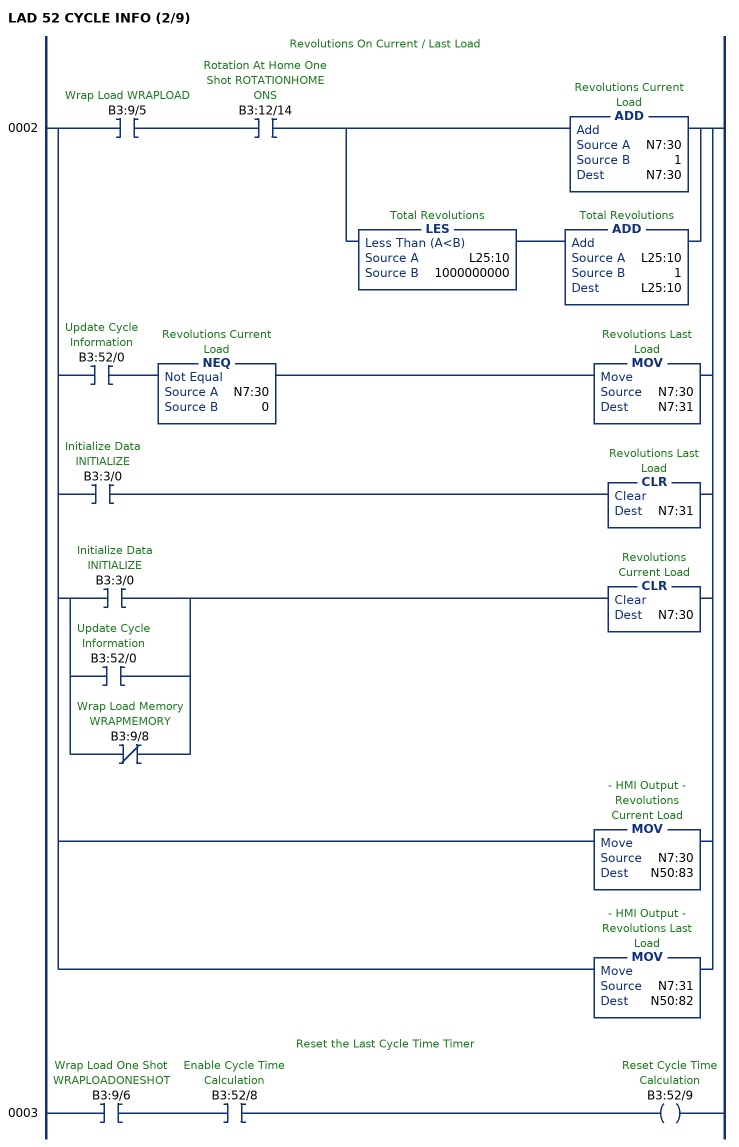
% Rung: 2 %
% Revolutions On Current / Last Load %
SOR BST XIC B3:9/5 XIC B3:12/14 BST ADD N7:30 1 N7:30 NXB LES L25:10 1000000000 ADD L25:10 1 L25:10 BND NXB XIC B3:52/0 NEQ N7:30 0 MOV N7:30 N7:31 NXB XIC B3:3/0 CLR N7:31 NXB BST XIC B3:3/0 NXB XIC B3:52/0 NXB XIO B3:9/8 BND CLR N7:30 NXB MOV N7:30 N50:83 NXB MOV N7:31 N50:82 BND EOR
%   B3:9/5  WRAPLOAD  "Wrap Load" %
%   B3:12/14  ROTATIONHOMEONS  "Rotation At Home One Shot" %
%   N7:30  "Revolutions Current Load" %
%   L25:10  "Total Revolutions" %
%   B3:52/0  "Update Cycle Information" %
%   N7:31  "Revolutions Last Load" %
%   B3:3/0  INITIALIZE  "Initialize Data" %
%   B3:9/8  WRAPMEMORY  "Wrap Load Memory" %
%   N50:83  "- HMI Output - Revolutions Current Load" %
%   N50:82  "- HMI Output - Revolutions Last Load" %
% Rung: 3 %
% Reset the Last Cycle Time Timer %
SOR XIC B3:9/6 XIC B3:52/8 OTE B3:52/9 EOR
%   B3:9/6  WRAPLOADONESHOT  "Wrap Load One Shot" %
%   B3:52/8  "Enable Cycle Time Calculation" %
%   B3:52/9  "Reset Cycle Time Calculation" %

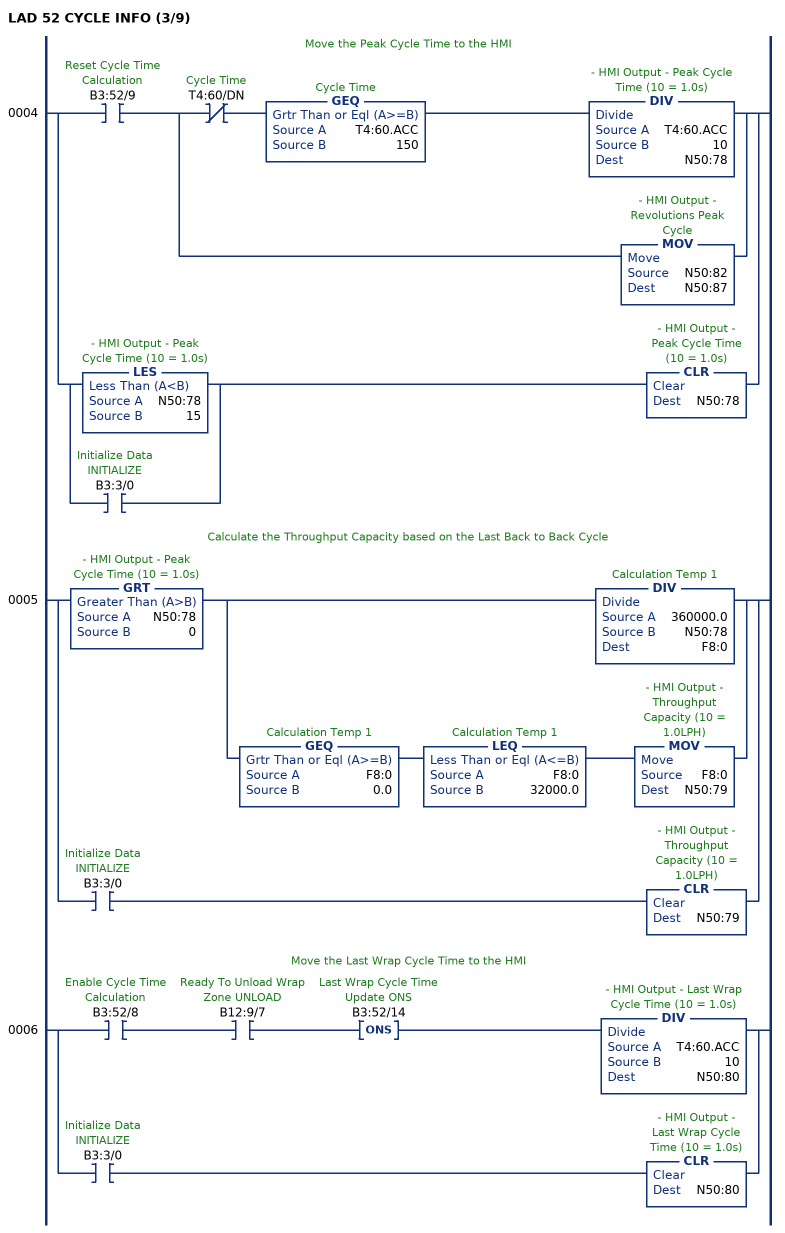
% Rung: 4 %
% Move the Peak Cycle Time to the HMI %
SOR BST XIC B3:52/9 BST XIO T4:60/DN GEQ T4:60.ACC 150 DIV T4:60.ACC 10 N50:78 NXB MOV N50:82 N50:87 BND NXB BST LES N50:78 15 NXB XIC B3:3/0 BND CLR N50:78 BND EOR
%   B3:52/9  "Reset Cycle Time Calculation" %
%   T4:60  "Cycle Time" %
%   N50:78  "- HMI Output - Peak Cycle Time (10 = 1.0s)" %
%   N50:82  "- HMI Output - Revolutions Last Load" %
%   N50:87  "- HMI Output - Revolutions Peak Cycle" %
%   B3:3/0  INITIALIZE  "Initialize Data" %
% Rung: 5 %
% Calculate the Throughput Capacity based on the Last Back to Back Cycle %
SOR BST GRT N50:78 0 BST DIV 360000.0 N50:78 F8:0 NXB GEQ F8:0 0.0 LEQ F8:0 32000.0 MOV F8:0 N50:79 BND NXB XIC B3:3/0 CLR N50:79 BND EOR
%   N50:78  "- HMI Output - Peak Cycle Time (10 = 1.0s)" %
%   F8:0  "Calculation Temp 1" %
%   N50:79  "- HMI Output - Throughput Capacity (10 = 1.0LPH)" %
%   B3:3/0  INITIALIZE  "Initialize Data" %
% Rung: 6 %
% Move the Last Wrap Cycle Time to the HMI %
SOR BST XIC B3:52/8 XIC B12:9/7 ONS B3:52/14 DIV T4:60.ACC 10 N50:80 NXB XIC B3:3/0 CLR N50:80 BND EOR
%   B3:52/8  "Enable Cycle Time Calculation" %
%   B12:9/7  UNLOAD  "Ready To Unload Wrap Zone" %
%   B3:52/14  "Last Wrap Cycle Time Update ONS" %
%   T4:60  "Cycle Time" %
%   N50:80  "- HMI Output - Last Wrap Cycle Time (10 = 1.0s)" %
%   B3:3/0  INITIALIZE  "Initialize Data" %

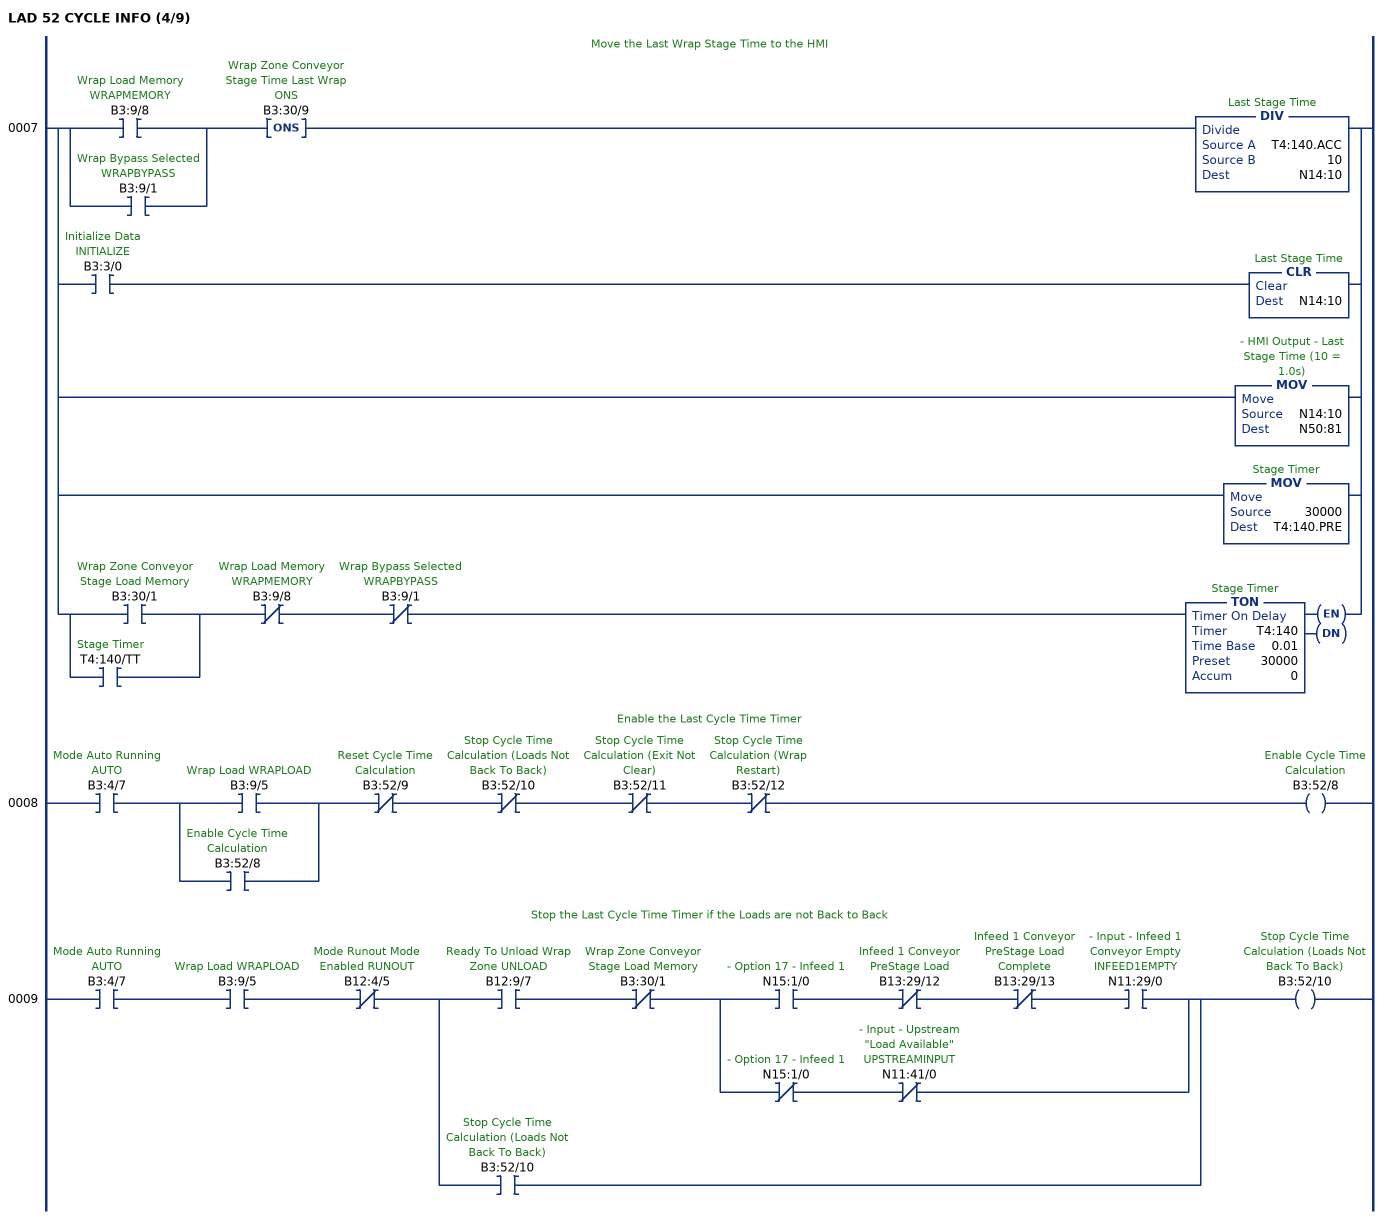
% Rung: 7 %
% Move the Last Wrap Stage Time to the HMI %
SOR BST BST XIC B3:9/8 NXB XIC B3:9/1 BND ONS B3:30/9 DIV T4:140.ACC 10 N14:10 NXB XIC B3:3/0 CLR N14:10 NXB MOV N14:10 N50:81 NXB MOV 30000 T4:140.PRE NXB BST XIC B3:30/1 NXB XIC T4:140/TT BND XIO B3:9/8 XIO B3:9/1 TON T4:140 0.01 30000 0 BND EOR
%   B3:9/8  WRAPMEMORY  "Wrap Load Memory" %
%   B3:9/1  WRAPBYPASS  "Wrap Bypass Selected" %
%   B3:30/9  "Wrap Zone Conveyor Stage Time Last Wrap ONS" %
%   T4:140  "Stage Timer" %
%   N14:10  "Last Stage Time" %
%   B3:3/0  INITIALIZE  "Initialize Data" %
%   N50:81  "- HMI Output - Last Stage Time (10 = 1.0s)" %
%   B3:30/1  "Wrap Zone Conveyor Stage Load Memory" %
% Rung: 8 %
% Enable the Last Cycle Time Timer %
SOR XIC B3:4/7 BST XIC B3:9/5 NXB XIC B3:52/8 BND XIO B3:52/9 XIO B3:52/10 XIO B3:52/11 XIO B3:52/12 OTE B3:52/8 EOR
%   B3:4/7  AUTO  "Mode Auto Running" %
%   B3:9/5  WRAPLOAD  "Wrap Load" %
%   B3:52/8  "Enable Cycle Time Calculation" %
%   B3:52/9  "Reset Cycle Time Calculation" %
%   B3:52/10  "Stop Cycle Time Calculation (Loads Not Back To Back)" %
%   B3:52/11  "Stop Cycle Time Calculation (Exit Not Clear)" %
%   B3:52/12  "Stop Cycle Time Calculation (Wrap Restart)" %
% Rung: 9 %
% Stop the Last Cycle Time Timer if the Loads are not Back to Back %
SOR XIC B3:4/7 XIC B3:9/5 XIO B12:4/5 BST XIC B12:9/7 XIO B3:30/1 BST XIC N15:1/0 XIO B13:29/12 XIO B13:29/13 XIC N11:29/0 NXB XIO N15:1/0 XIO N11:41/0 BND NXB XIC B3:52/10 BND OTE B3:52/10 EOR
%   B3:4/7  AUTO  "Mode Auto Running" %
%   B3:9/5  WRAPLOAD  "Wrap Load" %
%   B12:4/5  RUNOUT  "Mode Runout Mode Enabled" %
%   B12:9/7  UNLOAD  "Ready To Unload Wrap Zone" %
%   B3:30/1  "Wrap Zone Conveyor Stage Load Memory" %
%   N15:1/0  "- Option 17 - Infeed 1" %
%   B13:29/12  "Infeed 1 Conveyor PreStage Load" %
%   B13:29/13  "Infeed 1 Conveyor PreStage Load Complete" %
%   N11:29/0  INFEED1EMPTY  "- Input - Infeed 1 Conveyor Empty" %
%   N11:41/0  UPSTREAMINPUT  "- Input - Upstream "Load Available"" %
%   B3:52/10  "Stop Cycle Time Calculation (Loads Not Back To Back)" %

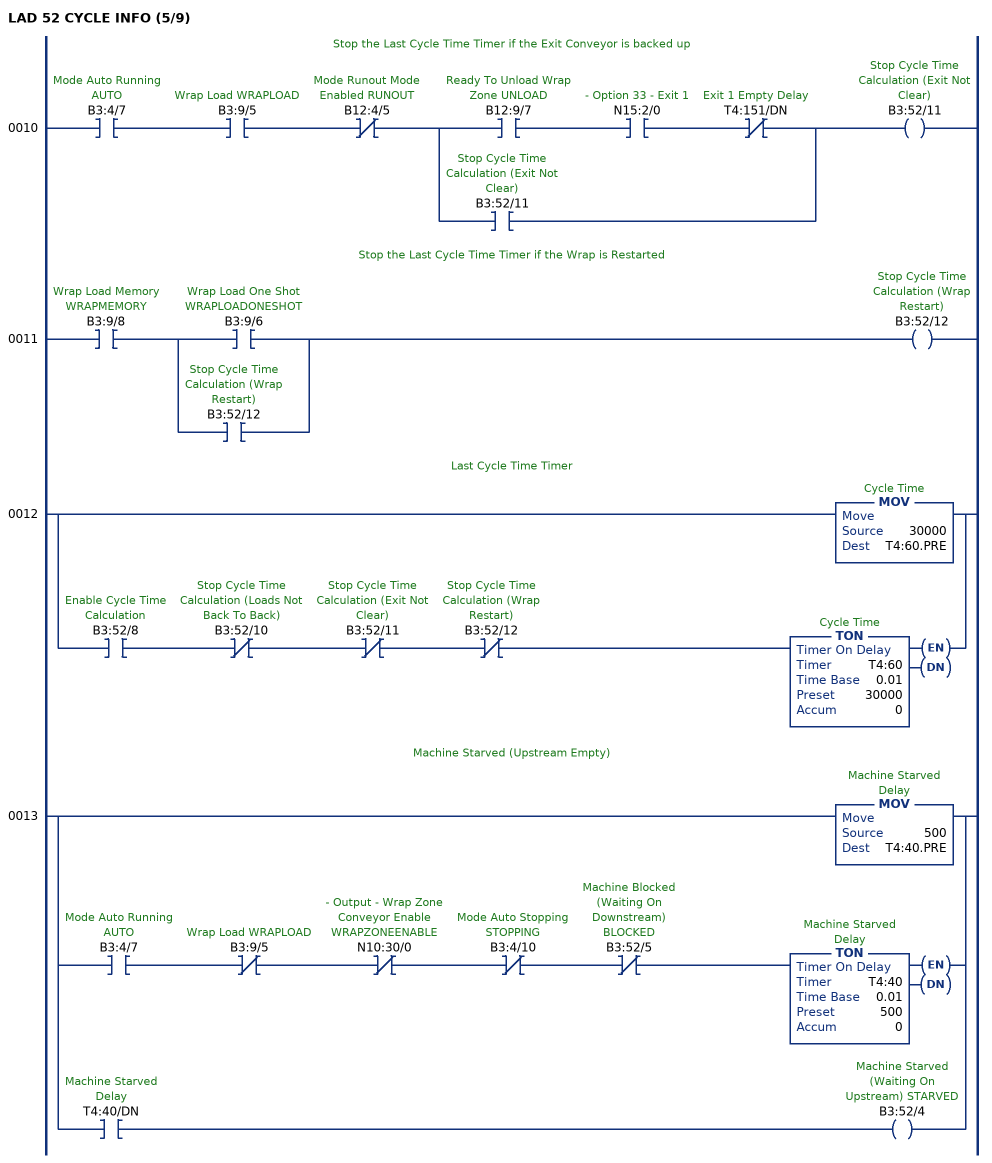
% Rung: 10 %
% Stop the Last Cycle Time Timer if the Exit Conveyor is backed up %
SOR XIC B3:4/7 XIC B3:9/5 XIO B12:4/5 BST XIC B12:9/7 XIC N15:2/0 XIO T4:151/DN NXB XIC B3:52/11 BND OTE B3:52/11 EOR
%   B3:4/7  AUTO  "Mode Auto Running" %
%   B3:9/5  WRAPLOAD  "Wrap Load" %
%   B12:4/5  RUNOUT  "Mode Runout Mode Enabled" %
%   B12:9/7  UNLOAD  "Ready To Unload Wrap Zone" %
%   N15:2/0  "- Option 33 - Exit 1" %
%   T4:151  "Exit 1 Empty Delay" %
%   B3:52/11  "Stop Cycle Time Calculation (Exit Not Clear)" %
% Rung: 11 %
% Stop the Last Cycle Time Timer if the Wrap is Restarted %
SOR XIC B3:9/8 BST XIC B3:9/6 NXB XIC B3:52/12 BND OTE B3:52/12 EOR
%   B3:9/8  WRAPMEMORY  "Wrap Load Memory" %
%   B3:9/6  WRAPLOADONESHOT  "Wrap Load One Shot" %
%   B3:52/12  "Stop Cycle Time Calculation (Wrap Restart)" %
% Rung: 12 %
% Last Cycle Time Timer %
SOR BST MOV 30000 T4:60.PRE NXB XIC B3:52/8 XIO B3:52/10 XIO B3:52/11 XIO B3:52/12 TON T4:60 0.01 30000 0 BND EOR
%   T4:60  "Cycle Time" %
%   B3:52/8  "Enable Cycle Time Calculation" %
%   B3:52/10  "Stop Cycle Time Calculation (Loads Not Back To Back)" %
%   B3:52/11  "Stop Cycle Time Calculation (Exit Not Clear)" %
%   B3:52/12  "Stop Cycle Time Calculation (Wrap Restart)" %
% Rung: 13 %
% Machine Starved (Upstream Empty) %
SOR BST MOV 500 T4:40.PRE NXB XIC B3:4/7 XIO B3:9/5 XIO N10:30/0 XIO B3:4/10 XIO B3:52/5 TON T4:40 0.01 500 0 NXB XIC T4:40/DN OTE B3:52/4 BND EOR
%   T4:40  "Machine Starved Delay" %
%   B3:4/7  AUTO  "Mode Auto Running" %
%   B3:9/5  WRAPLOAD  "Wrap Load" %
%   N10:30/0  WRAPZONEENABLE  "- Output - Wrap Zone Conveyor Enable" %
%   B3:4/10  STOPPING  "Mode Auto Stopping" %
%   B3:52/5  BLOCKED  "Machine Blocked (Waiting On Downstream)" %
%   B3:52/4  STARVED  "Machine Starved (Waiting On Upstream)" %

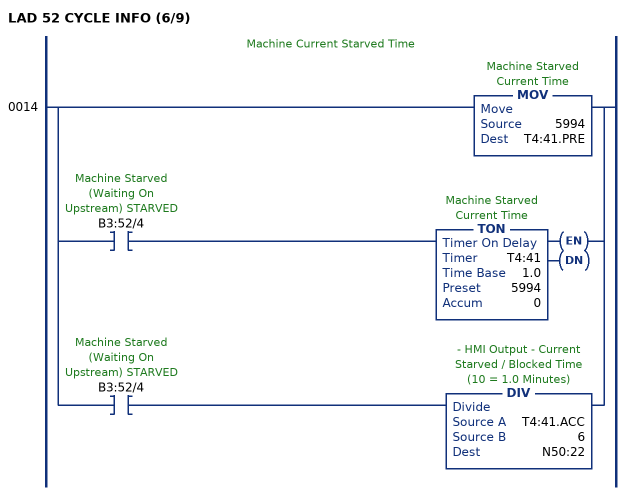
% Rung: 14 %
% Machine Current Starved Time %
SOR BST MOV 5994 T4:41.PRE NXB XIC B3:52/4 TON T4:41 1.0 5994 0 NXB XIC B3:52/4 DIV T4:41.ACC 6 N50:22 BND EOR
%   T4:41  "Machine Starved Current Time" %
%   B3:52/4  STARVED  "Machine Starved (Waiting On Upstream)" %
%   N50:22  "- HMI Output - Current Starved / Blocked Time (10 = 1.0 Minutes)" %

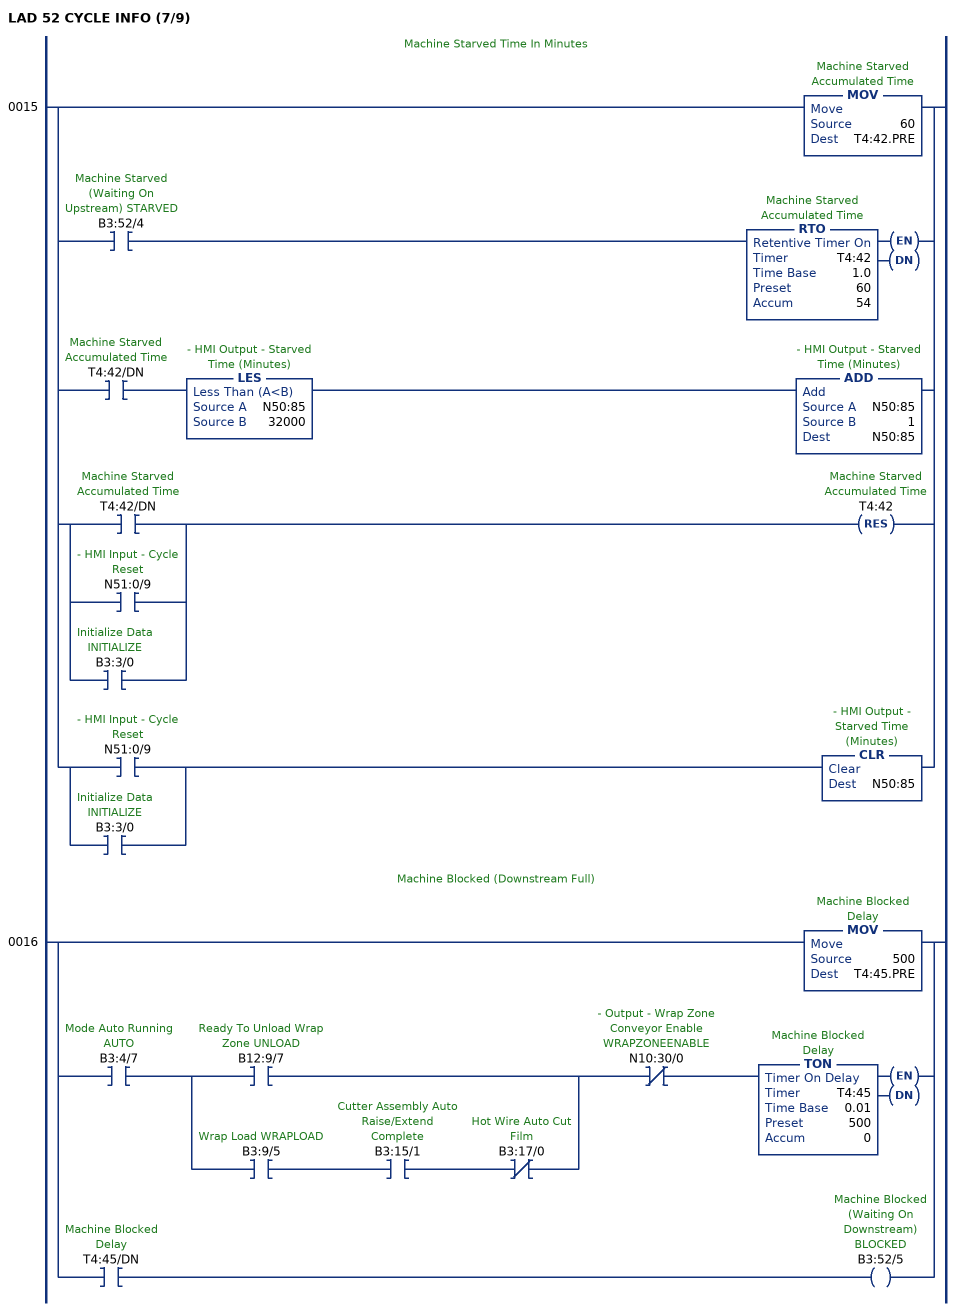
% Rung: 15 %
% Machine Starved Time In Minutes %
SOR BST MOV 60 T4:42.PRE NXB XIC B3:52/4 RTO T4:42 1.0 60 54 NXB XIC T4:42/DN LES N50:85 32000 ADD N50:85 1 N50:85 NXB BST XIC T4:42/DN NXB XIC N51:0/9 NXB XIC B3:3/0 BND RES T4:42 NXB BST XIC N51:0/9 NXB XIC B3:3/0 BND CLR N50:85 BND EOR
%   T4:42  "Machine Starved Accumulated Time" %
%   B3:52/4  STARVED  "Machine Starved (Waiting On Upstream)" %
%   N50:85  "- HMI Output - Starved Time (Minutes)" %
%   N51:0/9  "- HMI Input - Cycle Reset" %
%   B3:3/0  INITIALIZE  "Initialize Data" %
% Rung: 16 %
% Machine Blocked (Downstream Full) %
SOR BST MOV 500 T4:45.PRE NXB XIC B3:4/7 BST XIC B12:9/7 NXB XIC B3:9/5 XIC B3:15/1 XIO B3:17/0 BND XIO N10:30/0 TON T4:45 0.01 500 0 NXB XIC T4:45/DN OTE B3:52/5 BND EOR
%   T4:45  "Machine Blocked Delay" %
%   B3:4/7  AUTO  "Mode Auto Running" %
%   B12:9/7  UNLOAD  "Ready To Unload Wrap Zone" %
%   B3:9/5  WRAPLOAD  "Wrap Load" %
%   B3:15/1  "Cutter Assembly Auto Raise/Extend Complete" %
%   B3:17/0  "Hot Wire Auto Cut Film" %
%   N10:30/0  WRAPZONEENABLE  "- Output - Wrap Zone Conveyor Enable" %
%   B3:52/5  BLOCKED  "Machine Blocked (Waiting On Downstream)" %

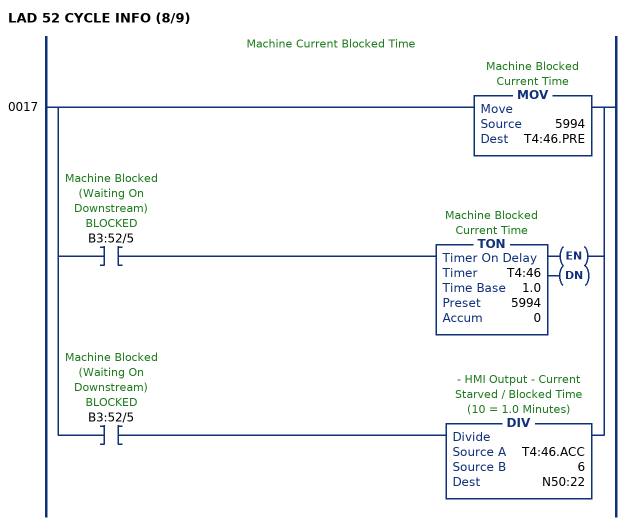
% Rung: 17 %
% Machine Current Blocked Time %
SOR BST MOV 5994 T4:46.PRE NXB XIC B3:52/5 TON T4:46 1.0 5994 0 NXB XIC B3:52/5 DIV T4:46.ACC 6 N50:22 BND EOR
%   T4:46  "Machine Blocked Current Time" %
%   B3:52/5  BLOCKED  "Machine Blocked (Waiting On Downstream)" %
%   N50:22  "- HMI Output - Current Starved / Blocked Time (10 = 1.0 Minutes)" %

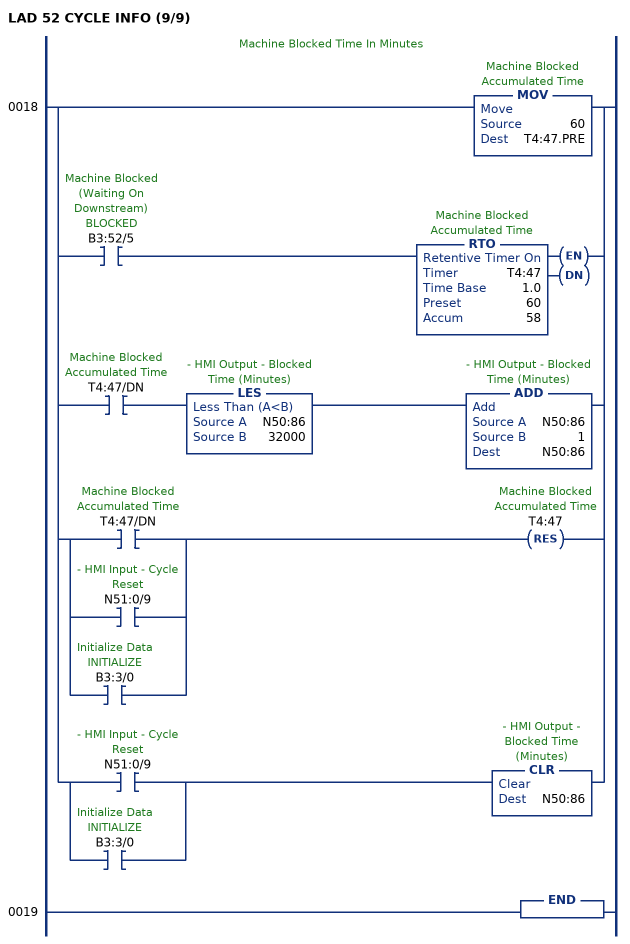
% Rung: 18 %
% Machine Blocked Time In Minutes %
SOR BST MOV 60 T4:47.PRE NXB XIC B3:52/5 RTO T4:47 1.0 60 58 NXB XIC T4:47/DN LES N50:86 32000 ADD N50:86 1 N50:86 NXB BST XIC T4:47/DN NXB XIC N51:0/9 NXB XIC B3:3/0 BND RES T4:47 NXB BST XIC N51:0/9 NXB XIC B3:3/0 BND CLR N50:86 BND EOR
%   T4:47  "Machine Blocked Accumulated Time" %
%   B3:52/5  BLOCKED  "Machine Blocked (Waiting On Downstream)" %
%   N50:86  "- HMI Output - Blocked Time (Minutes)" %
%   N51:0/9  "- HMI Input - Cycle Reset" %
%   B3:3/0  INITIALIZE  "Initialize Data" %
% Rung: 19 %
SOR END EOR

LADDER 98 "WARNINGS"
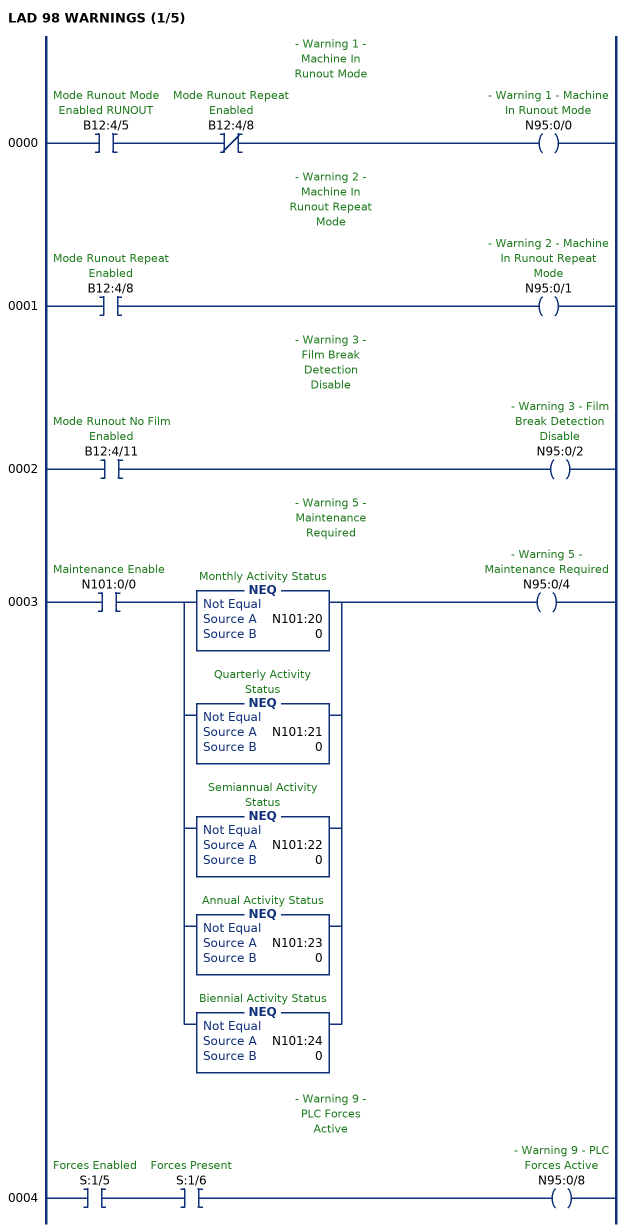
% Rung: 0 %
% - Warning 1 -
% Machine In
% Runout Mode %
SOR XIC B12:4/5 XIO B12:4/8 OTE N95:0/0 EOR
%   B12:4/5  RUNOUT  "Mode Runout Mode Enabled" %
%   B12:4/8  "Mode Runout Repeat Enabled" %
%   N95:0/0  "- Warning 1 - Machine In Runout Mode" %
% Rung: 1 %
% - Warning 2 -
% Machine In
% Runout Repeat
% Mode %
SOR XIC B12:4/8 OTE N95:0/1 EOR
%   B12:4/8  "Mode Runout Repeat Enabled" %
%   N95:0/1  "- Warning 2 - Machine In Runout Repeat Mode" %
% Rung: 2 %
% - Warning 3 -
% Film Break
% Detection
% Disable %
SOR XIC B12:4/11 OTE N95:0/2 EOR
%   B12:4/11  "Mode Runout No Film Enabled" %
%   N95:0/2  "- Warning 3 - Film Break Detection Disable" %
% Rung: 3 %
% - Warning 5 -
% Maintenance
% Required %
SOR XIC N101:0/0 BST NEQ N101:20 0 NXB NEQ N101:21 0 NXB NEQ N101:22 0 NXB NEQ N101:23 0 NXB NEQ N101:24 0 BND OTE N95:0/4 EOR
%   N101:0/0  "Maintenance Enable" %
%   N101:20  "Monthly Activity Status" %
%   N101:21  "Quarterly Activity Status" %
%   N101:22  "Semiannual Activity Status" %
%   N101:23  "Annual Activity Status" %
%   N101:24  "Biennial Activity Status" %
%   N95:0/4  "- Warning 5 - Maintenance Required" %
% Rung: 4 %
% - Warning 9 -
% PLC Forces
% Active %
SOR XIC S:1/5 XIC S:1/6 OTE N95:0/8 EOR
%   S:1/5  "Forces Enabled" %
%   S:1/6  "Forces Present" %
%   N95:0/8  "- Warning 9 - PLC Forces Active" %

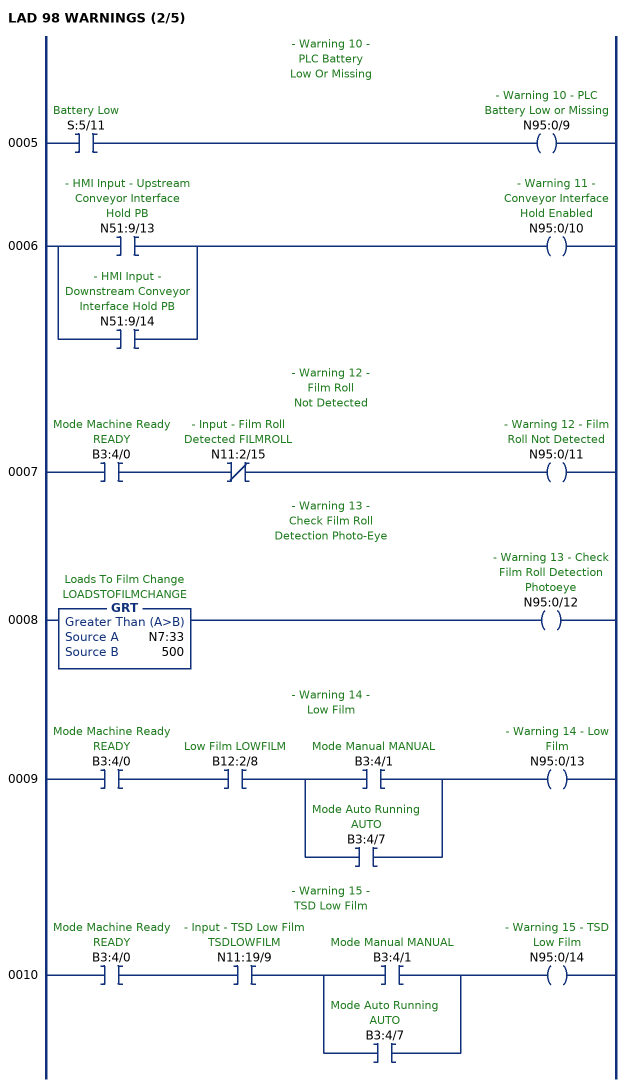
% Rung: 5 %
% - Warning 10 -
% PLC Battery
% Low Or Missing %
SOR XIC S:5/11 OTE N95:0/9 EOR
%   S:5/11  "Battery Low" %
%   N95:0/9  "- Warning 10 - PLC Battery Low or Missing" %
% Rung: 6 %
SOR BST XIC N51:9/13 NXB XIC N51:9/14 BND OTE N95:0/10 EOR
%   N51:9/13  "- HMI Input - Upstream Conveyor Interface Hold PB" %
%   N51:9/14  "- HMI Input - Downstream Conveyor Interface Hold PB" %
%   N95:0/10  "- Warning 11 - Conveyor Interface Hold Enabled" %
% Rung: 7 %
% - Warning 12 -
% Film Roll
% Not Detected %
SOR XIC B3:4/0 XIO N11:2/15 OTE N95:0/11 EOR
%   B3:4/0  READY  "Mode Machine Ready" %
%   N11:2/15  FILMROLL  "- Input - Film Roll Detected" %
%   N95:0/11  "- Warning 12 - Film Roll Not Detected" %
% Rung: 8 %
% - Warning 13 -
% Check Film Roll
% Detection Photo-Eye %
SOR GRT N7:33 500 OTE N95:0/12 EOR
%   N7:33  LOADSTOFILMCHANGE  "Loads To Film Change" %
%   N95:0/12  "- Warning 13 - Check Film Roll Detection Photoeye" %
% Rung: 9 %
% - Warning 14 -
% 
% Low Film %
SOR XIC B3:4/0 XIC B12:2/8 BST XIC B3:4/1 NXB XIC B3:4/7 BND OTE N95:0/13 EOR
%   B3:4/0  READY  "Mode Machine Ready" %
%   B12:2/8  LOWFILM  "Low Film" %
%   B3:4/1  MANUAL  "Mode Manual" %
%   B3:4/7  AUTO  "Mode Auto Running" %
%   N95:0/13  "- Warning 14 - Low Film" %
% Rung: 10 %
% - Warning 15 -
% 
% TSD Low Film %
SOR XIC B3:4/0 XIC N11:19/9 BST XIC B3:4/1 NXB XIC B3:4/7 BND OTE N95:0/14 EOR
%   B3:4/0  READY  "Mode Machine Ready" %
%   N11:19/9  TSDLOWFILM  "- Input - TSD Low Film" %
%   B3:4/1  MANUAL  "Mode Manual" %
%   B3:4/7  AUTO  "Mode Auto Running" %
%   N95:0/14  "- Warning 15 - TSD Low Film" %

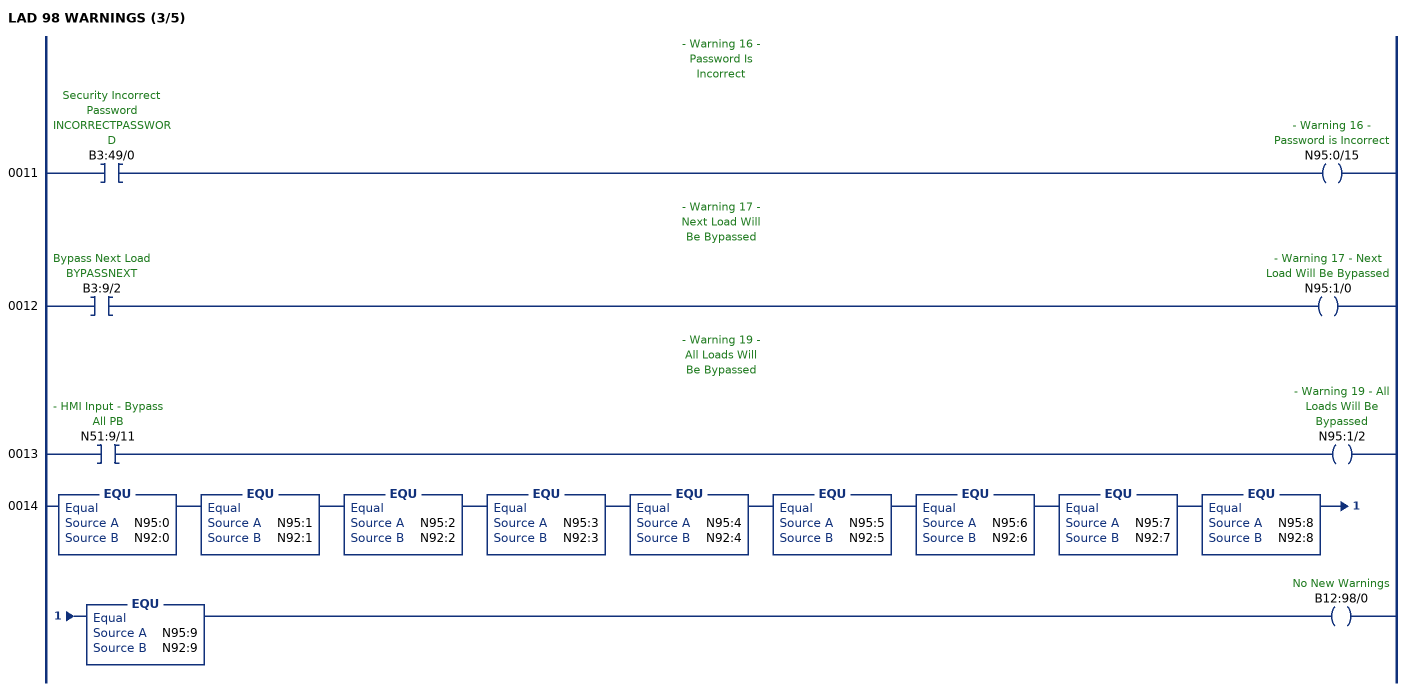
% Rung: 11 %
% - Warning 16 -
% Password Is
% Incorrect %
SOR XIC B3:49/0 OTE N95:0/15 EOR
%   B3:49/0  INCORRECTPASSWORD  "Security Incorrect Password" %
%   N95:0/15  "- Warning 16 - Password is Incorrect" %
% Rung: 12 %
% - Warning 17 -
% Next Load Will
% Be Bypassed %
SOR XIC B3:9/2 OTE N95:1/0 EOR
%   B3:9/2  BYPASSNEXT  "Bypass Next Load" %
%   N95:1/0  "- Warning 17 - Next Load Will Be Bypassed" %
% Rung: 13 %
% - Warning 19 -
% All Loads Will
% Be Bypassed %
SOR XIC N51:9/11 OTE N95:1/2 EOR
%   N51:9/11  "- HMI Input - Bypass All PB" %
%   N95:1/2  "- Warning 19 - All Loads Will Be Bypassed" %
% Rung: 14 %
SOR EQU N95:0 N92:0 EQU N95:1 N92:1 EQU N95:2 N92:2 EQU N95:3 N92:3 EQU N95:4 N92:4 EQU N95:5 N92:5 EQU N95:6 N92:6 EQU N95:7 N92:7 EQU N95:8 N92:8 EQU N95:9 N92:9 OTE B12:98/0 EOR
%   B12:98/0  "No New Warnings" %

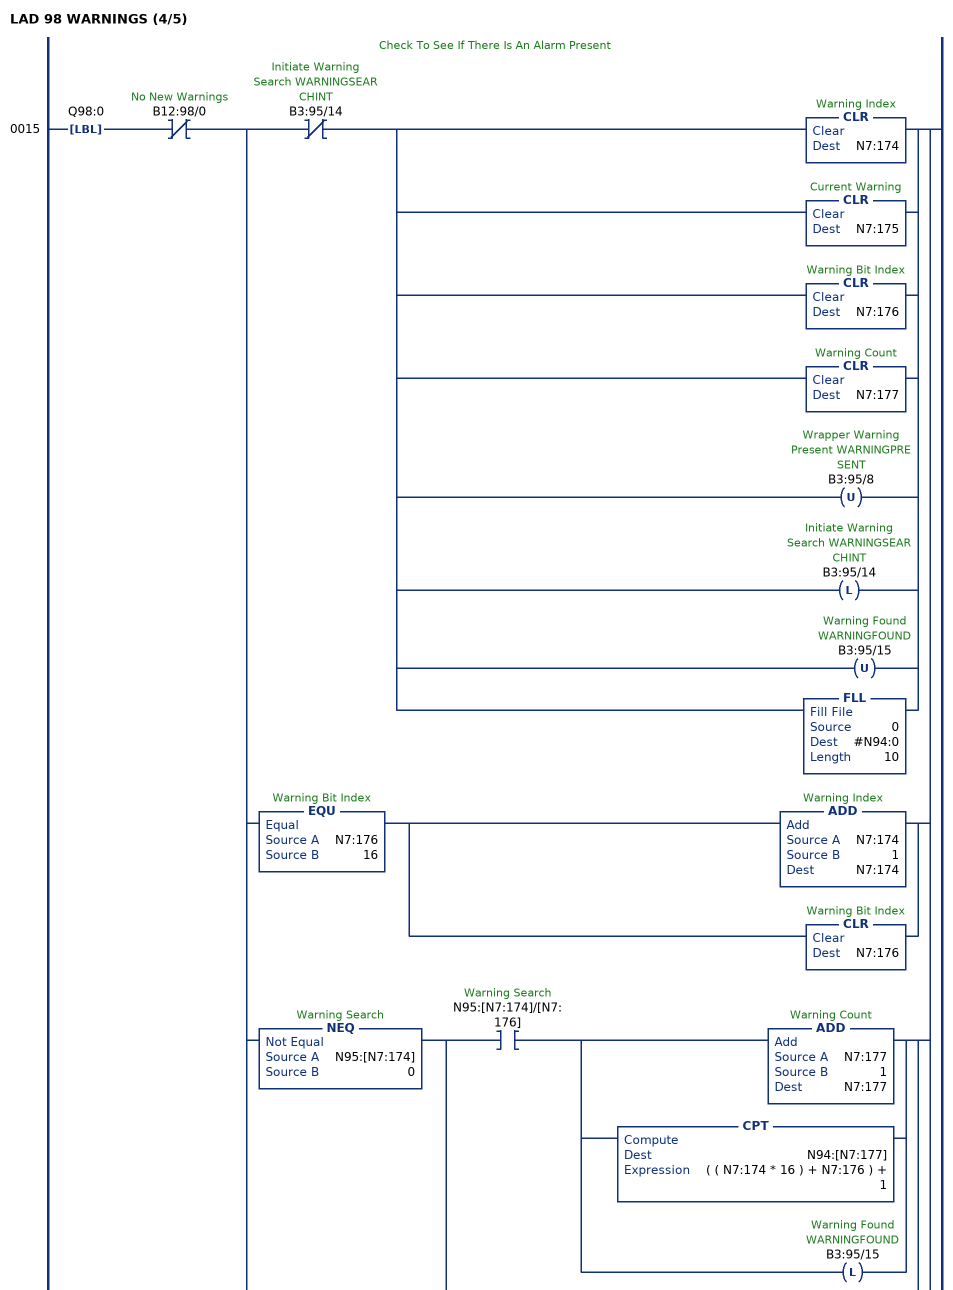

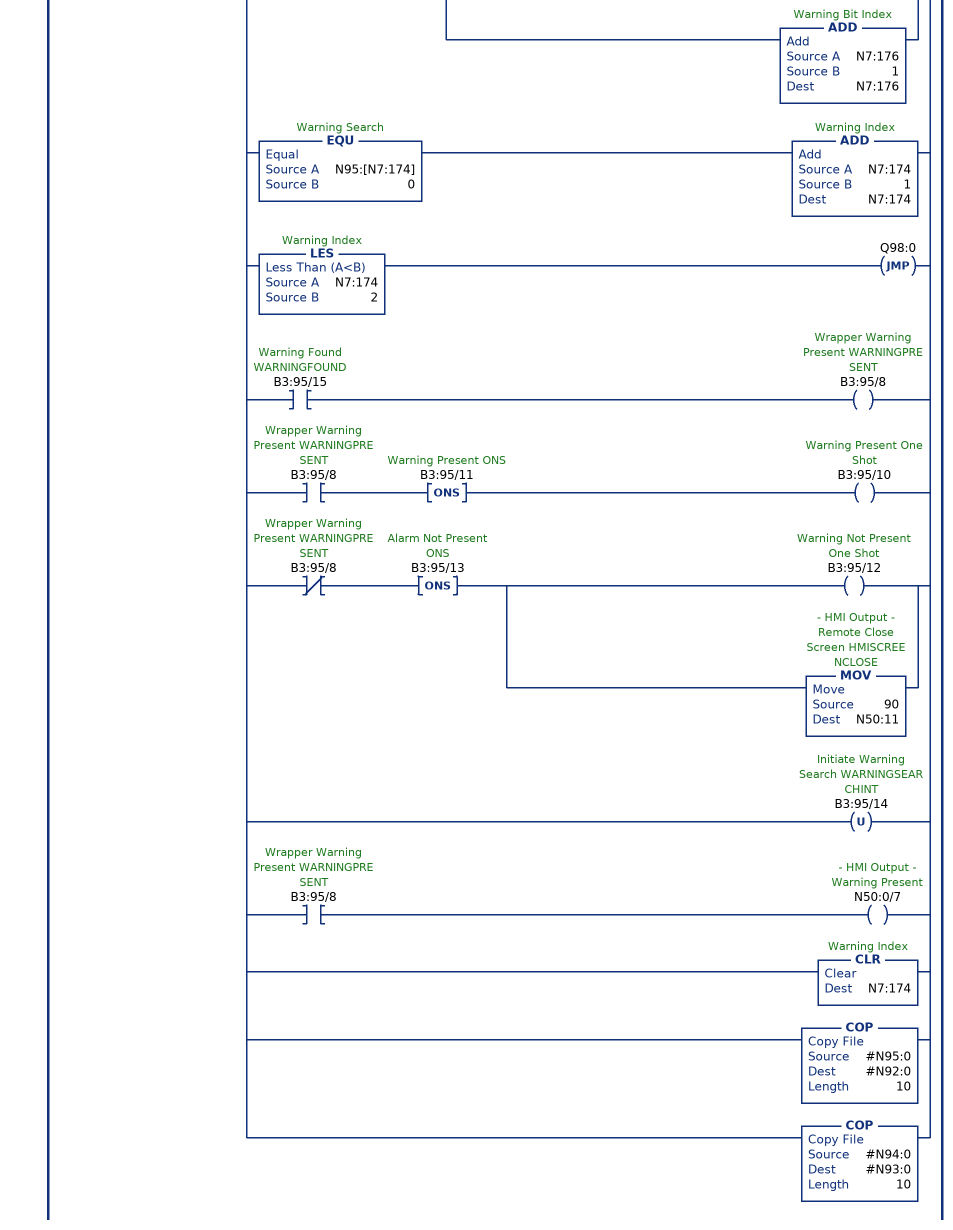
% Rung: 15 %
% Check To See If There Is An Alarm Present %
SOR LBL Q98:0 XIO B12:98/0 BST XIO B3:95/14 BST CLR N7:174 NXB CLR N7:175 NXB CLR N7:176 NXB CLR N7:177 NXB OTU B3:95/8 NXB OTL B3:95/14 NXB OTU B3:95/15 NXB FLL 0 #N94:0 10 BND NXB EQU N7:176 16 BST ADD N7:174 1 N7:174 NXB CLR N7:176 BND NXB NEQ N95:[N7:174] 0 BST XIC N95:[N7:174]/[N7:176] BST ADD N7:177 1 N7:177 NXB CPT N94:[N7:177] " ( ( N7:174 * 16 ) + N7:176 ) + 1 " NXB OTL B3:95/15 BND NXB ADD N7:176 1 N7:176 BND NXB EQU N95:[N7:174] 0 ADD N7:174 1 N7:174 NXB LES N7:174 2 JMP Q98:0 NXB XIC B3:95/15 OTE B3:95/8 NXB XIC B3:95/8 ONS B3:95/11 OTE B3:95/10 NXB XIO B3:95/8 ONS B3:95/13 BST OTE B3:95/12 NXB MOV 90 N50:11 BND NXB OTU B3:95/14 NXB XIC B3:95/8 OTE N50:0/7 NXB CLR N7:174 NXB COP #N95:0 #N92:0 10 NXB COP #N94:0 #N93:0 10 BND EOR
%   B12:98/0  "No New Warnings" %
%   B3:95/14  WARNINGSEARCHINT  "Initiate Warning Search" %
%   N7:174  "Warning Index" %
%   N7:175  "Current Warning" %
%   N7:176  "Warning Bit Index" %
%   N7:177  "Warning Count" %
%   B3:95/8  WARNINGPRESENT  "Wrapper Warning Present" %
%   B3:95/15  WARNINGFOUND  "Warning Found" %
%   N95:[N7:174]  "Warning Search" %
%   N95:[N7:174]/[N7:176]  "Warning Search" %
%   B3:95/11  "Warning Present ONS" %
%   B3:95/10  "Warning Present One Shot" %
%   B3:95/13  "Alarm Not Present ONS" %
%   B3:95/12  "Warning Not Present One Shot" %
%   N50:11  HMISCREENCLOSE  "- HMI Output - Remote Close Screen" %
%   N50:0/7  "- HMI Output - Warning Present" %

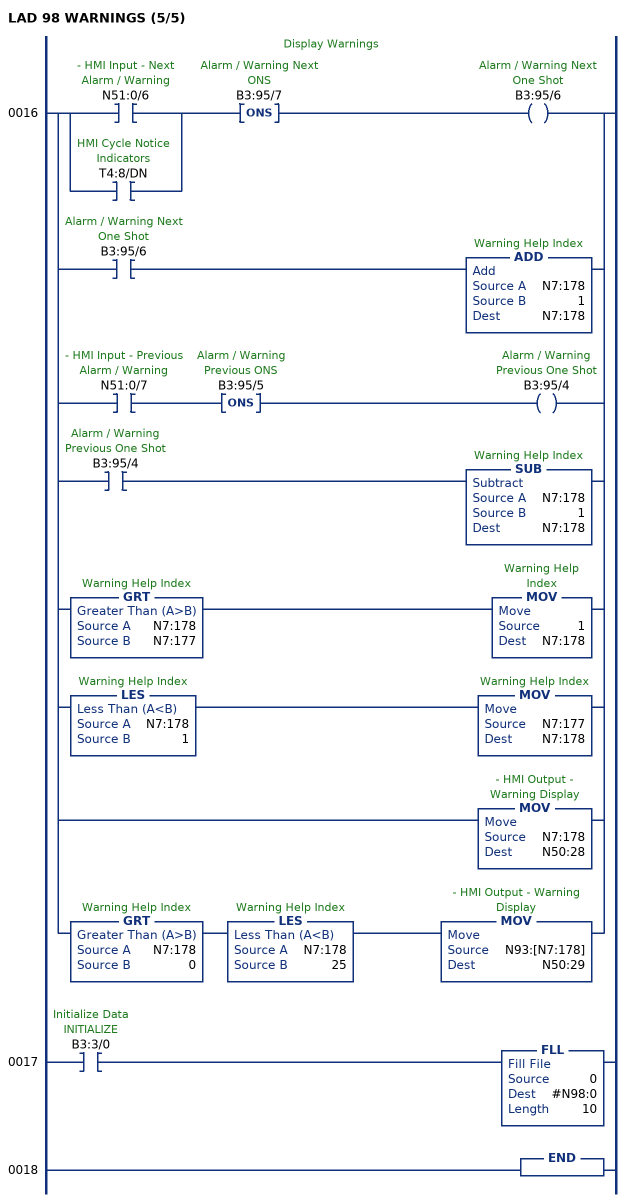
% Rung: 16 %
% Display Warnings %
SOR BST BST XIC N51:0/6 NXB XIC T4:8/DN BND ONS B3:95/7 OTE B3:95/6 NXB XIC B3:95/6 ADD N7:178 1 N7:178 NXB XIC N51:0/7 ONS B3:95/5 OTE B3:95/4 NXB XIC B3:95/4 SUB N7:178 1 N7:178 NXB GRT N7:178 N7:177 MOV 1 N7:178 NXB LES N7:178 1 MOV N7:177 N7:178 NXB MOV N7:178 N50:28 NXB GRT N7:178 0 LES N7:178 25 MOV N93:[N7:178] N50:29 BND EOR
%   N51:0/6  "- HMI Input - Next Alarm / Warning" %
%   T4:8  "HMI Cycle Notice Indicators" %
%   B3:95/7  "Alarm / Warning Next ONS" %
%   B3:95/6  "Alarm / Warning Next One Shot" %
%   N7:178  "Warning Help Index" %
%   N51:0/7  "- HMI Input - Previous Alarm / Warning" %
%   B3:95/5  "Alarm / Warning Previous ONS" %
%   B3:95/4  "Alarm / Warning Previous One Shot" %
%   N7:177  "Warning Count" %
%   N50:28  "- HMI Output - Warning Display" %
%   N50:29  "- HMI Output - Warning Display" %
% Rung: 17 %
SOR XIC B3:3/0 FLL 0 #N98:0 10 EOR
%   B3:3/0  INITIALIZE  "Initialize Data" %
% Rung: 18 %
SOR END EOR

LADDER 99 "MESSAGES"
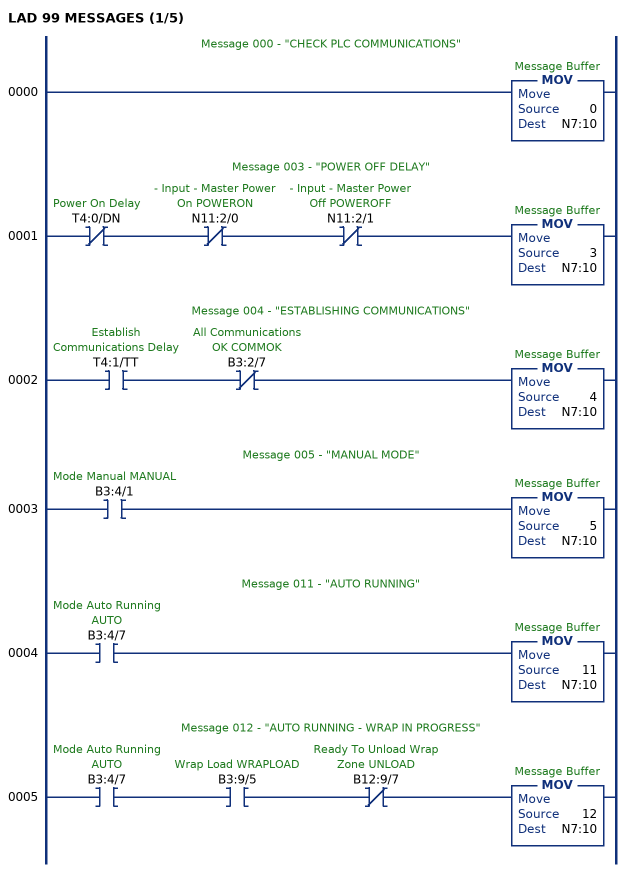
% Rung: 0 %
% Message 000 - "CHECK PLC COMMUNICATIONS" %
SOR MOV 0 N7:10 EOR
%   N7:10  "Message Buffer" %
% Rung: 1 %
% Message 003 - "POWER OFF DELAY" %
SOR XIO T4:0/DN XIO N11:2/0 XIO N11:2/1 MOV 3 N7:10 EOR
%   T4:0  "Power On Delay" %
%   N11:2/0  POWERON  "- Input - Master Power On" %
%   N11:2/1  POWEROFF  "- Input - Master Power Off" %
%   N7:10  "Message Buffer" %
% Rung: 2 %
% Message 004 - "ESTABLISHING COMMUNICATIONS" %
SOR XIC T4:1/TT XIO B3:2/7 MOV 4 N7:10 EOR
%   T4:1  "Establish Communications Delay" %
%   B3:2/7  COMMOK  "All Communications OK" %
%   N7:10  "Message Buffer" %
% Rung: 3 %
% Message 005 - "MANUAL MODE" %
SOR XIC B3:4/1 MOV 5 N7:10 EOR
%   B3:4/1  MANUAL  "Mode Manual" %
%   N7:10  "Message Buffer" %
% Rung: 4 %
% Message 011 - "AUTO RUNNING" %
SOR XIC B3:4/7 MOV 11 N7:10 EOR
%   B3:4/7  AUTO  "Mode Auto Running" %
%   N7:10  "Message Buffer" %
% Rung: 5 %
% Message 012 - "AUTO RUNNING - WRAP IN PROGRESS" %
SOR XIC B3:4/7 XIC B3:9/5 XIO B12:9/7 MOV 12 N7:10 EOR
%   B3:4/7  AUTO  "Mode Auto Running" %
%   B3:9/5  WRAPLOAD  "Wrap Load" %
%   B12:9/7  UNLOAD  "Ready To Unload Wrap Zone" %
%   N7:10  "Message Buffer" %

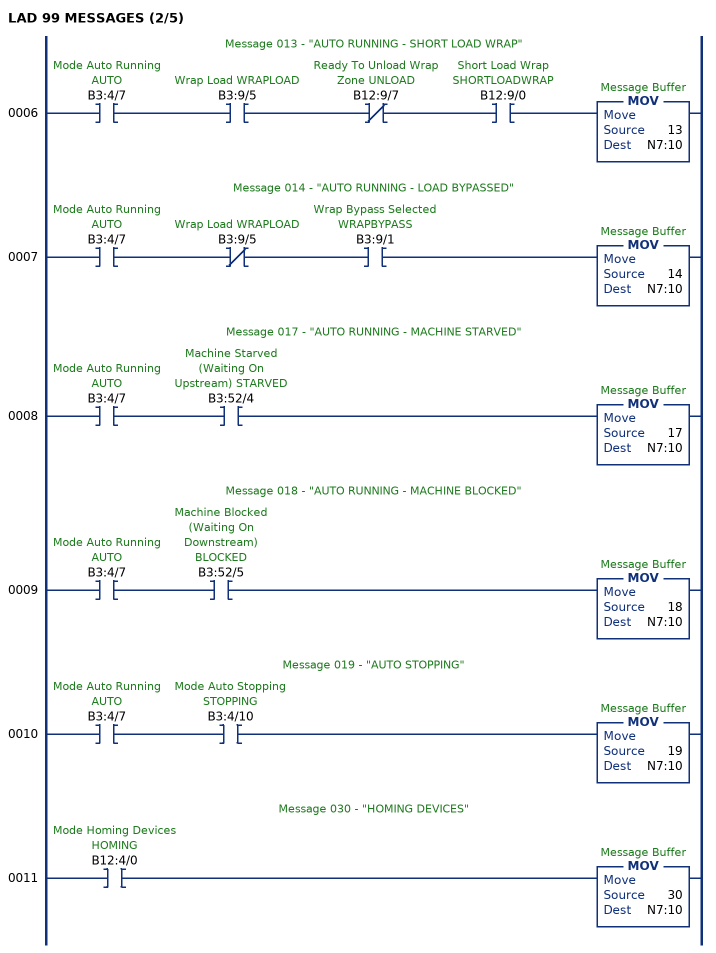
% Rung: 6 %
% Message 013 - "AUTO RUNNING - SHORT LOAD WRAP" %
SOR XIC B3:4/7 XIC B3:9/5 XIO B12:9/7 XIC B12:9/0 MOV 13 N7:10 EOR
%   B3:4/7  AUTO  "Mode Auto Running" %
%   B3:9/5  WRAPLOAD  "Wrap Load" %
%   B12:9/7  UNLOAD  "Ready To Unload Wrap Zone" %
%   B12:9/0  SHORTLOADWRAP  "Short Load Wrap" %
%   N7:10  "Message Buffer" %
% Rung: 7 %
% Message 014 - "AUTO RUNNING - LOAD BYPASSED" %
SOR XIC B3:4/7 XIO B3:9/5 XIC B3:9/1 MOV 14 N7:10 EOR
%   B3:4/7  AUTO  "Mode Auto Running" %
%   B3:9/5  WRAPLOAD  "Wrap Load" %
%   B3:9/1  WRAPBYPASS  "Wrap Bypass Selected" %
%   N7:10  "Message Buffer" %
% Rung: 8 %
% Message 017 - "AUTO RUNNING - MACHINE STARVED" %
SOR XIC B3:4/7 XIC B3:52/4 MOV 17 N7:10 EOR
%   B3:4/7  AUTO  "Mode Auto Running" %
%   B3:52/4  STARVED  "Machine Starved (Waiting On Upstream)" %
%   N7:10  "Message Buffer" %
% Rung: 9 %
% Message 018 - "AUTO RUNNING - MACHINE BLOCKED" %
SOR XIC B3:4/7 XIC B3:52/5 MOV 18 N7:10 EOR
%   B3:4/7  AUTO  "Mode Auto Running" %
%   B3:52/5  BLOCKED  "Machine Blocked (Waiting On Downstream)" %
%   N7:10  "Message Buffer" %
% Rung: 10 %
% Message 019 - "AUTO STOPPING" %
SOR XIC B3:4/7 XIC B3:4/10 MOV 19 N7:10 EOR
%   B3:4/7  AUTO  "Mode Auto Running" %
%   B3:4/10  STOPPING  "Mode Auto Stopping" %
%   N7:10  "Message Buffer" %
% Rung: 11 %
% Message 030 - "HOMING DEVICES" %
SOR XIC B12:4/0 MOV 30 N7:10 EOR
%   B12:4/0  HOMING  "Mode Homing Devices" %
%   N7:10  "Message Buffer" %

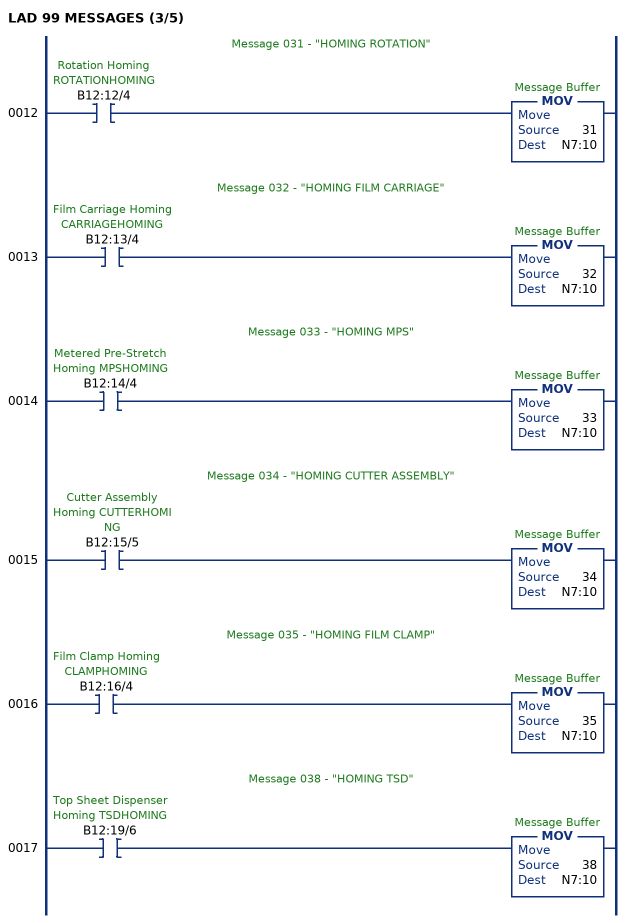
% Rung: 12 %
% Message 031 - "HOMING ROTATION" %
SOR XIC B12:12/4 MOV 31 N7:10 EOR
%   B12:12/4  ROTATIONHOMING  "Rotation Homing" %
%   N7:10  "Message Buffer" %
% Rung: 13 %
% Message 032 - "HOMING FILM CARRIAGE" %
SOR XIC B12:13/4 MOV 32 N7:10 EOR
%   B12:13/4  CARRIAGEHOMING  "Film Carriage Homing" %
%   N7:10  "Message Buffer" %
% Rung: 14 %
% Message 033 - "HOMING MPS" %
SOR XIC B12:14/4 MOV 33 N7:10 EOR
%   B12:14/4  MPSHOMING  "Metered Pre-Stretch Homing" %
%   N7:10  "Message Buffer" %
% Rung: 15 %
% Message 034 - "HOMING CUTTER ASSEMBLY" %
SOR XIC B12:15/5 MOV 34 N7:10 EOR
%   B12:15/5  CUTTERHOMING  "Cutter Assembly Homing" %
%   N7:10  "Message Buffer" %
% Rung: 16 %
% Message 035 - "HOMING FILM CLAMP" %
SOR XIC B12:16/4 MOV 35 N7:10 EOR
%   B12:16/4  CLAMPHOMING  "Film Clamp Homing" %
%   N7:10  "Message Buffer" %
% Rung: 17 %
% Message 038 - "HOMING TSD" %
SOR XIC B12:19/6 MOV 38 N7:10 EOR
%   B12:19/6  TSDHOMING  "Top Sheet Dispenser Homing" %
%   N7:10  "Message Buffer" %

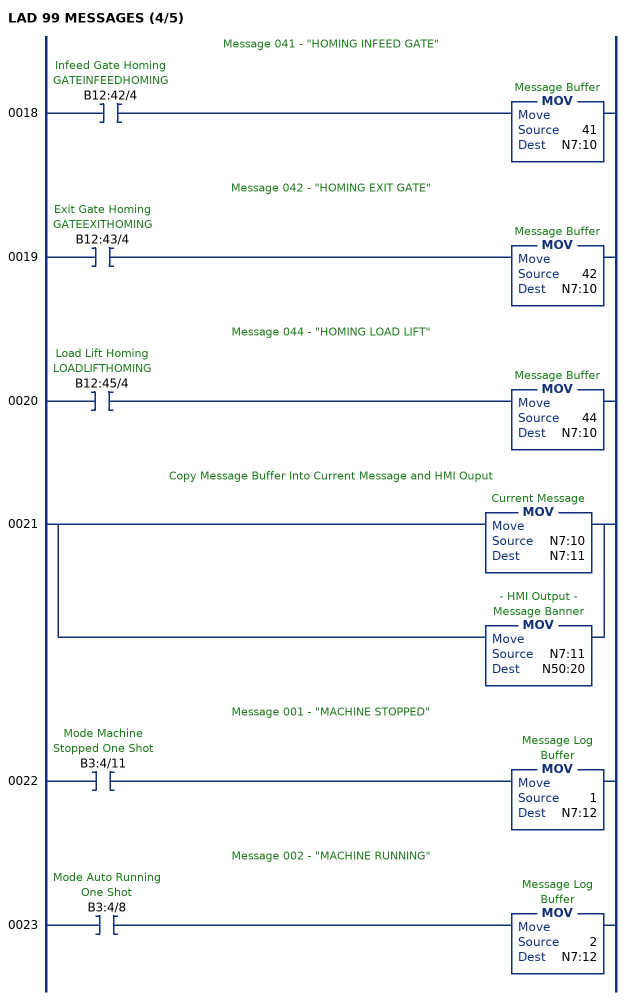
% Rung: 18 %
% Message 041 - "HOMING INFEED GATE" %
SOR XIC B12:42/4 MOV 41 N7:10 EOR
%   B12:42/4  GATEINFEEDHOMING  "Infeed Gate Homing" %
%   N7:10  "Message Buffer" %
% Rung: 19 %
% Message 042 - "HOMING EXIT GATE" %
SOR XIC B12:43/4 MOV 42 N7:10 EOR
%   B12:43/4  GATEEXITHOMING  "Exit Gate Homing" %
%   N7:10  "Message Buffer" %
% Rung: 20 %
% Message 044 - "HOMING LOAD LIFT" %
SOR XIC B12:45/4 MOV 44 N7:10 EOR
%   B12:45/4  LOADLIFTHOMING  "Load Lift Homing" %
%   N7:10  "Message Buffer" %
% Rung: 21 %
% Copy Message Buffer Into Current Message and HMI Ouput %
SOR BST MOV N7:10 N7:11 NXB MOV N7:11 N50:20 BND EOR
%   N7:10  "Message Buffer" %
%   N7:11  "Current Message" %
%   N50:20  "- HMI Output - Message Banner" %
% Rung: 22 %
% Message 001 - "MACHINE STOPPED" %
SOR XIC B3:4/11 MOV 1 N7:12 EOR
%   B3:4/11  "Mode Machine Stopped One Shot" %
%   N7:12  "Message Log Buffer" %
% Rung: 23 %
% Message 002 - "MACHINE RUNNING" %
SOR XIC B3:4/8 MOV 2 N7:12 EOR
%   B3:4/8  "Mode Auto Running One Shot" %
%   N7:12  "Message Log Buffer" %

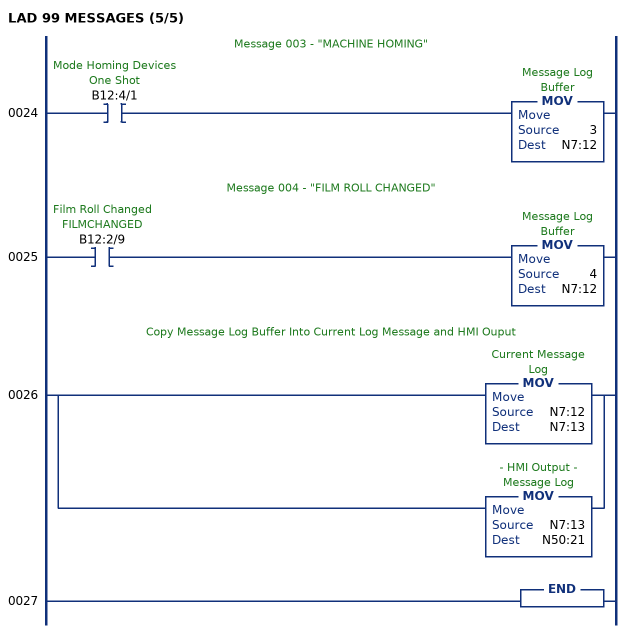
% Rung: 24 %
% Message 003 - "MACHINE HOMING" %
SOR XIC B12:4/1 MOV 3 N7:12 EOR
%   B12:4/1  "Mode Homing Devices One Shot" %
%   N7:12  "Message Log Buffer" %
% Rung: 25 %
% Message 004 - "FILM ROLL CHANGED" %
SOR XIC B12:2/9 MOV 4 N7:12 EOR
%   B12:2/9  FILMCHANGED  "Film Roll Changed" %
%   N7:12  "Message Log Buffer" %
% Rung: 26 %
% Copy Message Log Buffer Into Current Log Message and HMI Ouput %
SOR BST MOV N7:12 N7:13 NXB MOV N7:13 N50:21 BND EOR
%   N7:12  "Message Log Buffer" %
%   N7:13  "Current Message Log" %
%   N50:21  "- HMI Output - Message Log" %
% Rung: 27 %
SOR END EOR

LADDER 100 "ALARMS"
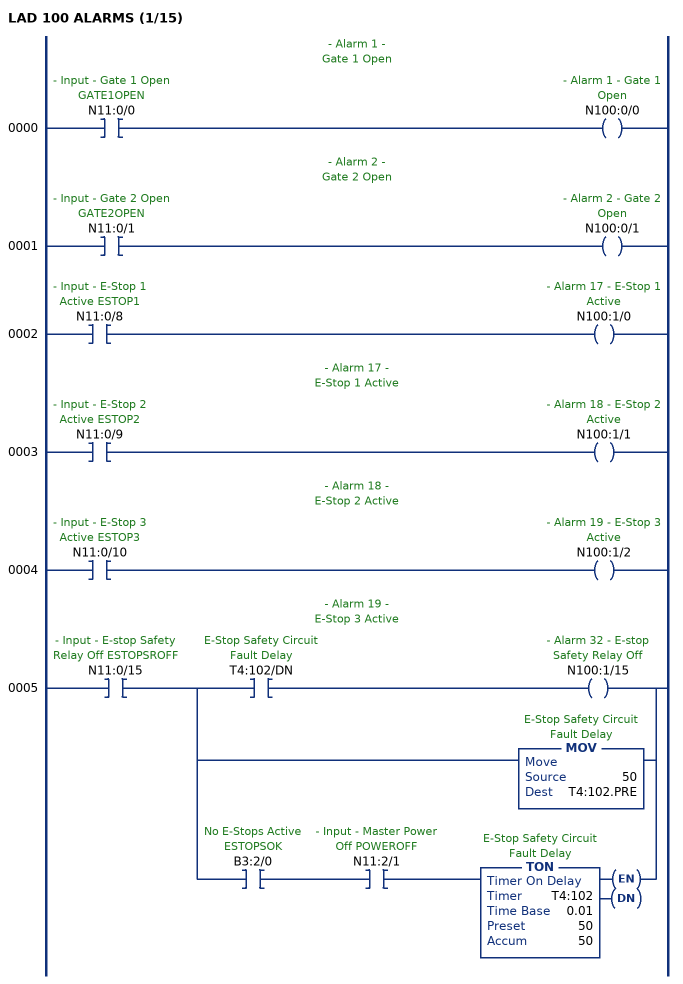
% Rung: 0 %
% - Alarm 1 -
% 
% Gate 1 Open %
SOR XIC N11:0/0 OTE N100:0/0 EOR
%   N11:0/0  GATE1OPEN  "- Input - Gate 1 Open" %
%   N100:0/0  "- Alarm 1 - Gate 1 Open" %
% Rung: 1 %
% - Alarm 2 -
% 
% Gate 2 Open %
SOR XIC N11:0/1 OTE N100:0/1 EOR
%   N11:0/1  GATE2OPEN  "- Input - Gate 2 Open" %
%   N100:0/1  "- Alarm 2 - Gate 2 Open" %
% Rung: 2 %
SOR XIC N11:0/8 OTE N100:1/0 EOR
%   N11:0/8  ESTOP1  "- Input - E-Stop 1 Active" %
%   N100:1/0  "- Alarm 17 - E-Stop 1 Active" %
% Rung: 3 %
% - Alarm 17 -
% 
% E-Stop 1 Active %
SOR XIC N11:0/9 OTE N100:1/1 EOR
%   N11:0/9  ESTOP2  "- Input - E-Stop 2 Active" %
%   N100:1/1  "- Alarm 18 - E-Stop 2 Active" %
% Rung: 4 %
% - Alarm 18 -
% 
% E-Stop 2 Active %
SOR XIC N11:0/10 OTE N100:1/2 EOR
%   N11:0/10  ESTOP3  "- Input - E-Stop 3 Active" %
%   N100:1/2  "- Alarm 19 - E-Stop 3 Active" %
% Rung: 5 %
% - Alarm 19 -
% 
% E-Stop 3 Active %
SOR XIC N11:0/15 BST XIC T4:102/DN OTE N100:1/15 NXB MOV 50 T4:102.PRE NXB XIC B3:2/0 XIC N11:2/1 TON T4:102 0.01 50 50 BND EOR
%   N11:0/15  ESTOPSROFF  "- Input - E-stop Safety Relay Off" %
%   T4:102  "E-Stop Safety Circuit Fault Delay" %
%   N100:1/15  "- Alarm 32 - E-stop Safety Relay Off" %
%   B3:2/0  ESTOPSOK  "No E-Stops Active" %
%   N11:2/1  POWEROFF  "- Input - Master Power Off" %

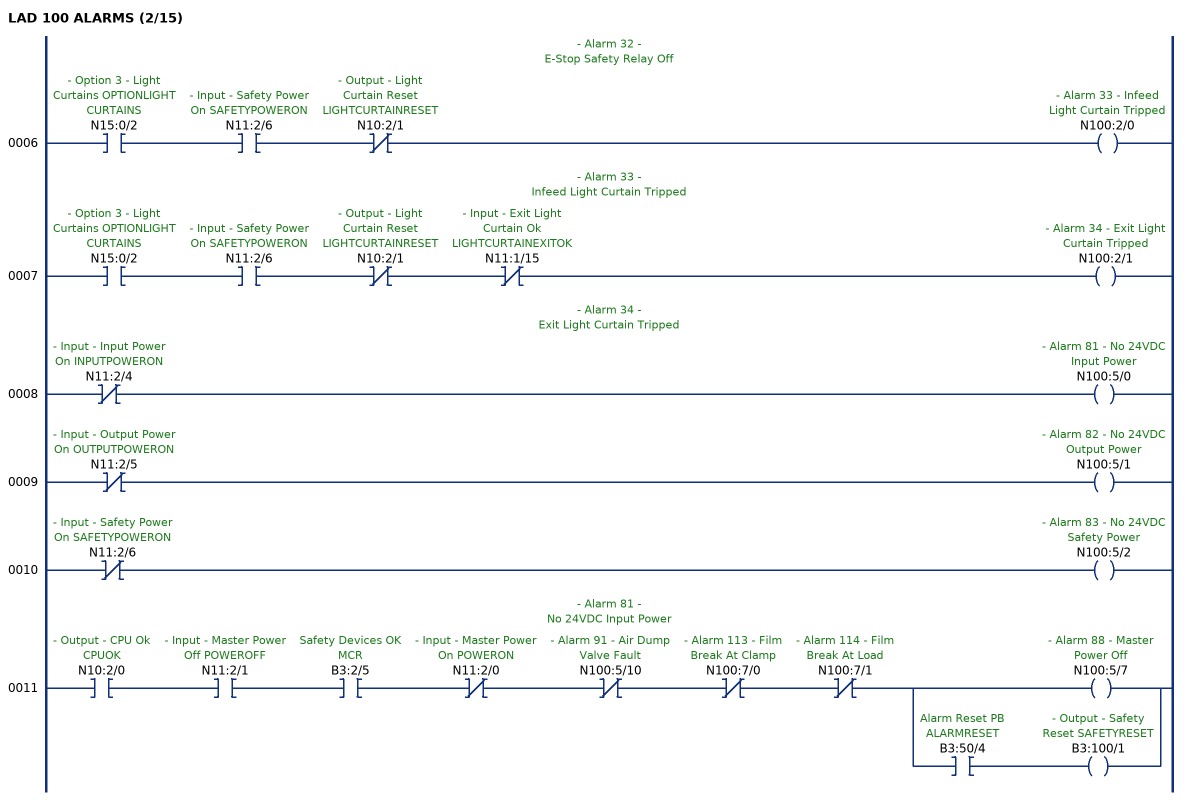
% Rung: 6 %
% - Alarm 32 -
% 
% E-Stop Safety Relay Off %
SOR XIC N15:0/2 XIC N11:2/6 XIO N10:2/1 OTE N100:2/0 EOR
%   N15:0/2  OPTIONLIGHTCURTAINS  "- Option 3 - Light Curtains" %
%   N11:2/6  SAFETYPOWERON  "- Input - Safety Power On" %
%   N10:2/1  LIGHTCURTAINRESET  "- Output - Light Curtain Reset" %
%   N100:2/0  "- Alarm 33 - Infeed Light Curtain Tripped" %
% Rung: 7 %
% - Alarm 33 -
% 
% Infeed Light Curtain Tripped %
SOR XIC N15:0/2 XIC N11:2/6 XIO N10:2/1 XIO N11:1/15 OTE N100:2/1 EOR
%   N15:0/2  OPTIONLIGHTCURTAINS  "- Option 3 - Light Curtains" %
%   N11:2/6  SAFETYPOWERON  "- Input - Safety Power On" %
%   N10:2/1  LIGHTCURTAINRESET  "- Output - Light Curtain Reset" %
%   N11:1/15  LIGHTCURTAINEXITOK  "- Input - Exit Light Curtain Ok" %
%   N100:2/1  "- Alarm 34 - Exit Light Curtain Tripped" %
% Rung: 8 %
% - Alarm 34 -
% 
% Exit Light Curtain Tripped %
SOR XIO N11:2/4 OTE N100:5/0 EOR
%   N11:2/4  INPUTPOWERON  "- Input - Input Power On" %
%   N100:5/0  "- Alarm 81 - No 24VDC Input Power" %
% Rung: 9 %
SOR XIO N11:2/5 OTE N100:5/1 EOR
%   N11:2/5  OUTPUTPOWERON  "- Input - Output Power On" %
%   N100:5/1  "- Alarm 82 - No 24VDC Output Power" %
% Rung: 10 %
SOR XIO N11:2/6 OTE N100:5/2 EOR
%   N11:2/6  SAFETYPOWERON  "- Input - Safety Power On" %
%   N100:5/2  "- Alarm 83 - No 24VDC Safety Power" %
% Rung: 11 %
% - Alarm 81 -
% 
% No 24VDC Input Power %
SOR XIC N10:2/0 XIC N11:2/1 XIC B3:2/5 XIO N11:2/0 XIO N100:5/10 XIO N100:7/0 XIO N100:7/1 BST OTE N100:5/7 NXB XIC B3:50/4 OTE B3:100/1 BND EOR
%   N10:2/0  CPUOK  "- Output - CPU Ok" %
%   N11:2/1  POWEROFF  "- Input - Master Power Off" %
%   B3:2/5  MCR  "Safety Devices OK" %
%   N11:2/0  POWERON  "- Input - Master Power On" %
%   N100:5/10  "- Alarm 91 - Air Dump Valve Fault" %
%   N100:7/0  "- Alarm 113 - Film Break At Clamp" %
%   N100:7/1  "- Alarm 114 - Film Break At Load" %
%   N100:5/7  "- Alarm 88 - Master Power Off" %
%   B3:50/4  ALARMRESET  "Alarm Reset PB" %
%   B3:100/1  SAFETYRESET  "- Output - Safety Reset" %

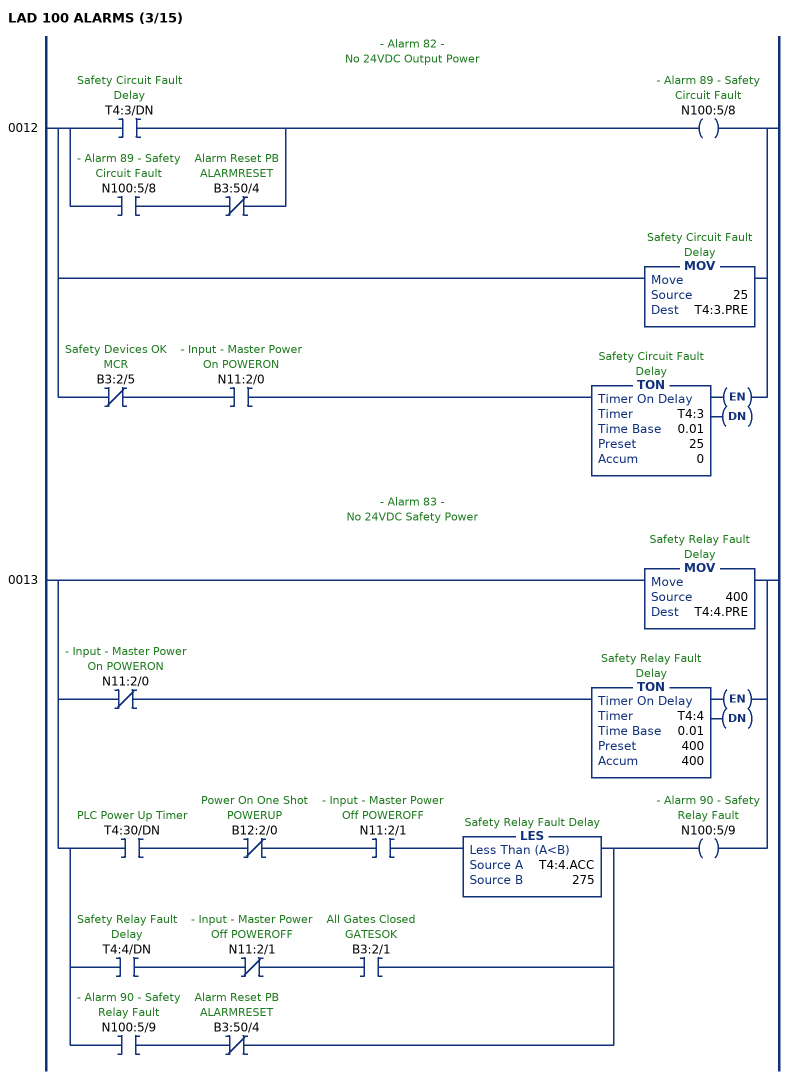
% Rung: 12 %
% - Alarm 82 -
% 
% No 24VDC Output Power %
SOR BST BST XIC T4:3/DN NXB XIC N100:5/8 XIO B3:50/4 BND OTE N100:5/8 NXB MOV 25 T4:3.PRE NXB XIO B3:2/5 XIC N11:2/0 TON T4:3 0.01 25 0 BND EOR
%   T4:3  "Safety Circuit Fault Delay" %
%   N100:5/8  "- Alarm 89 - Safety Circuit Fault" %
%   B3:50/4  ALARMRESET  "Alarm Reset PB" %
%   B3:2/5  MCR  "Safety Devices OK" %
%   N11:2/0  POWERON  "- Input - Master Power On" %
% Rung: 13 %
% - Alarm 83 -
% 
% No 24VDC Safety Power %
SOR BST MOV 400 T4:4.PRE NXB XIO N11:2/0 TON T4:4 0.01 400 400 NXB BST XIC T4:30/DN XIO B12:2/0 XIC N11:2/1 LES T4:4.ACC 275 NXB XIC T4:4/DN XIO N11:2/1 XIC B3:2/1 NXB XIC N100:5/9 XIO B3:50/4 BND OTE N100:5/9 BND EOR
%   T4:4  "Safety Relay Fault Delay" %
%   N11:2/0  POWERON  "- Input - Master Power On" %
%   T4:30  "PLC Power Up Timer" %
%   B12:2/0  POWERUP  "Power On One Shot" %
%   N11:2/1  POWEROFF  "- Input - Master Power Off" %
%   B3:2/1  GATESOK  "All Gates Closed" %
%   N100:5/9  "- Alarm 90 - Safety Relay Fault" %
%   B3:50/4  ALARMRESET  "Alarm Reset PB" %

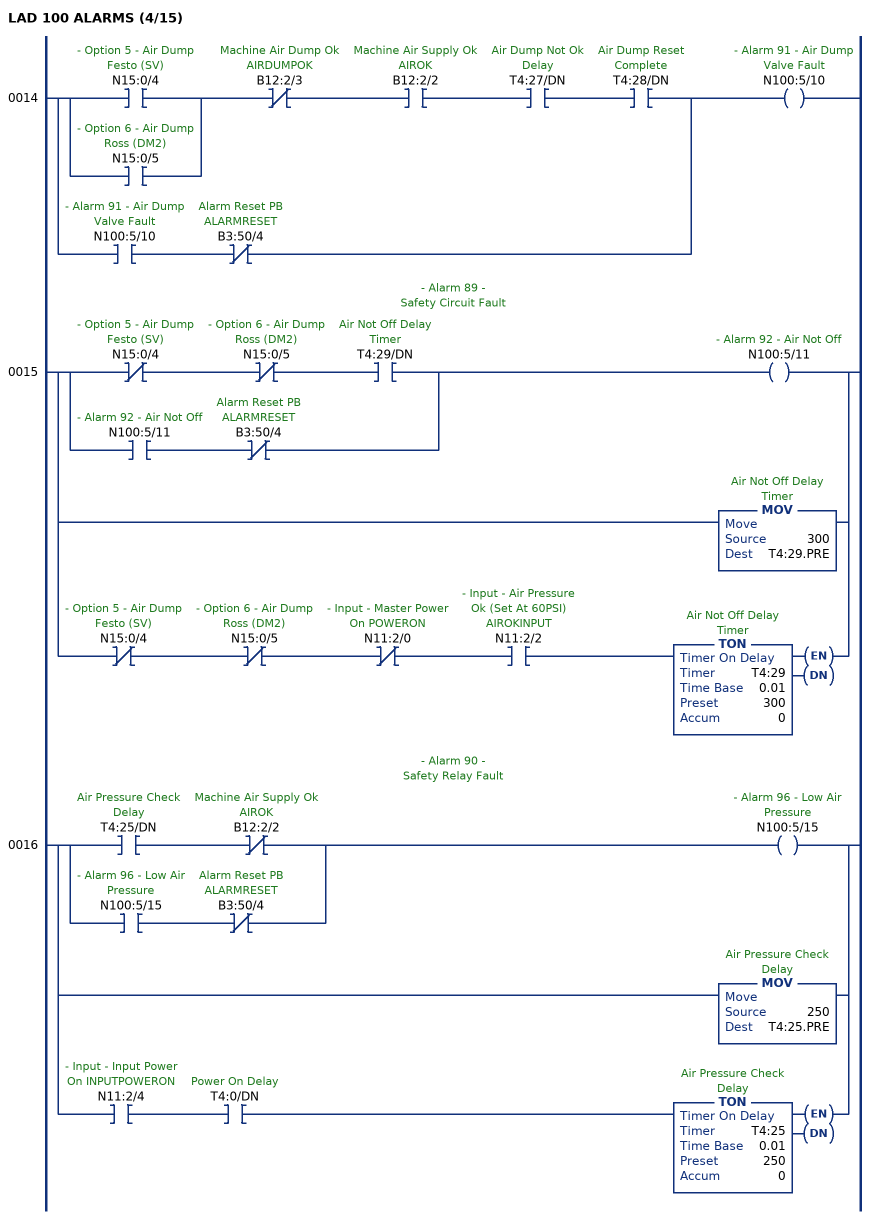
% Rung: 14 %
SOR BST BST XIC N15:0/4 NXB XIC N15:0/5 BND XIO B12:2/3 XIC B12:2/2 XIC T4:27/DN XIC T4:28/DN NXB XIC N100:5/10 XIO B3:50/4 BND OTE N100:5/10 EOR
%   N15:0/4  "- Option 5 - Air Dump Festo (SV)" %
%   N15:0/5  "- Option 6 - Air Dump Ross (DM2)" %
%   B12:2/3  AIRDUMPOK  "Machine Air Dump Ok" %
%   B12:2/2  AIROK  "Machine Air Supply Ok" %
%   T4:27  "Air Dump Not Ok Delay" %
%   T4:28  "Air Dump Reset Complete" %
%   N100:5/10  "- Alarm 91 - Air Dump Valve Fault" %
%   B3:50/4  ALARMRESET  "Alarm Reset PB" %
% Rung: 15 %
% - Alarm 89 -
% 
% Safety Circuit Fault %
SOR BST BST XIO N15:0/4 XIO N15:0/5 XIC T4:29/DN NXB XIC N100:5/11 XIO B3:50/4 BND OTE N100:5/11 NXB MOV 300 T4:29.PRE NXB XIO N15:0/4 XIO N15:0/5 XIO N11:2/0 XIC N11:2/2 TON T4:29 0.01 300 0 BND EOR
%   N15:0/4  "- Option 5 - Air Dump Festo (SV)" %
%   N15:0/5  "- Option 6 - Air Dump Ross (DM2)" %
%   T4:29  "Air Not Off Delay Timer" %
%   N100:5/11  "- Alarm 92 - Air Not Off" %
%   B3:50/4  ALARMRESET  "Alarm Reset PB" %
%   N11:2/0  POWERON  "- Input - Master Power On" %
%   N11:2/2  AIROKINPUT  "- Input - Air Pressure Ok (Set At 60PSI)" %
% Rung: 16 %
% - Alarm 90 -
% 
% Safety Relay Fault %
SOR BST BST XIC T4:25/DN XIO B12:2/2 NXB XIC N100:5/15 XIO B3:50/4 BND OTE N100:5/15 NXB MOV 250 T4:25.PRE NXB XIC N11:2/4 XIC T4:0/DN TON T4:25 0.01 250 0 BND EOR
%   T4:25  "Air Pressure Check Delay" %
%   B12:2/2  AIROK  "Machine Air Supply Ok" %
%   N100:5/15  "- Alarm 96 - Low Air Pressure" %
%   B3:50/4  ALARMRESET  "Alarm Reset PB" %
%   N11:2/4  INPUTPOWERON  "- Input - Input Power On" %
%   T4:0  "Power On Delay" %

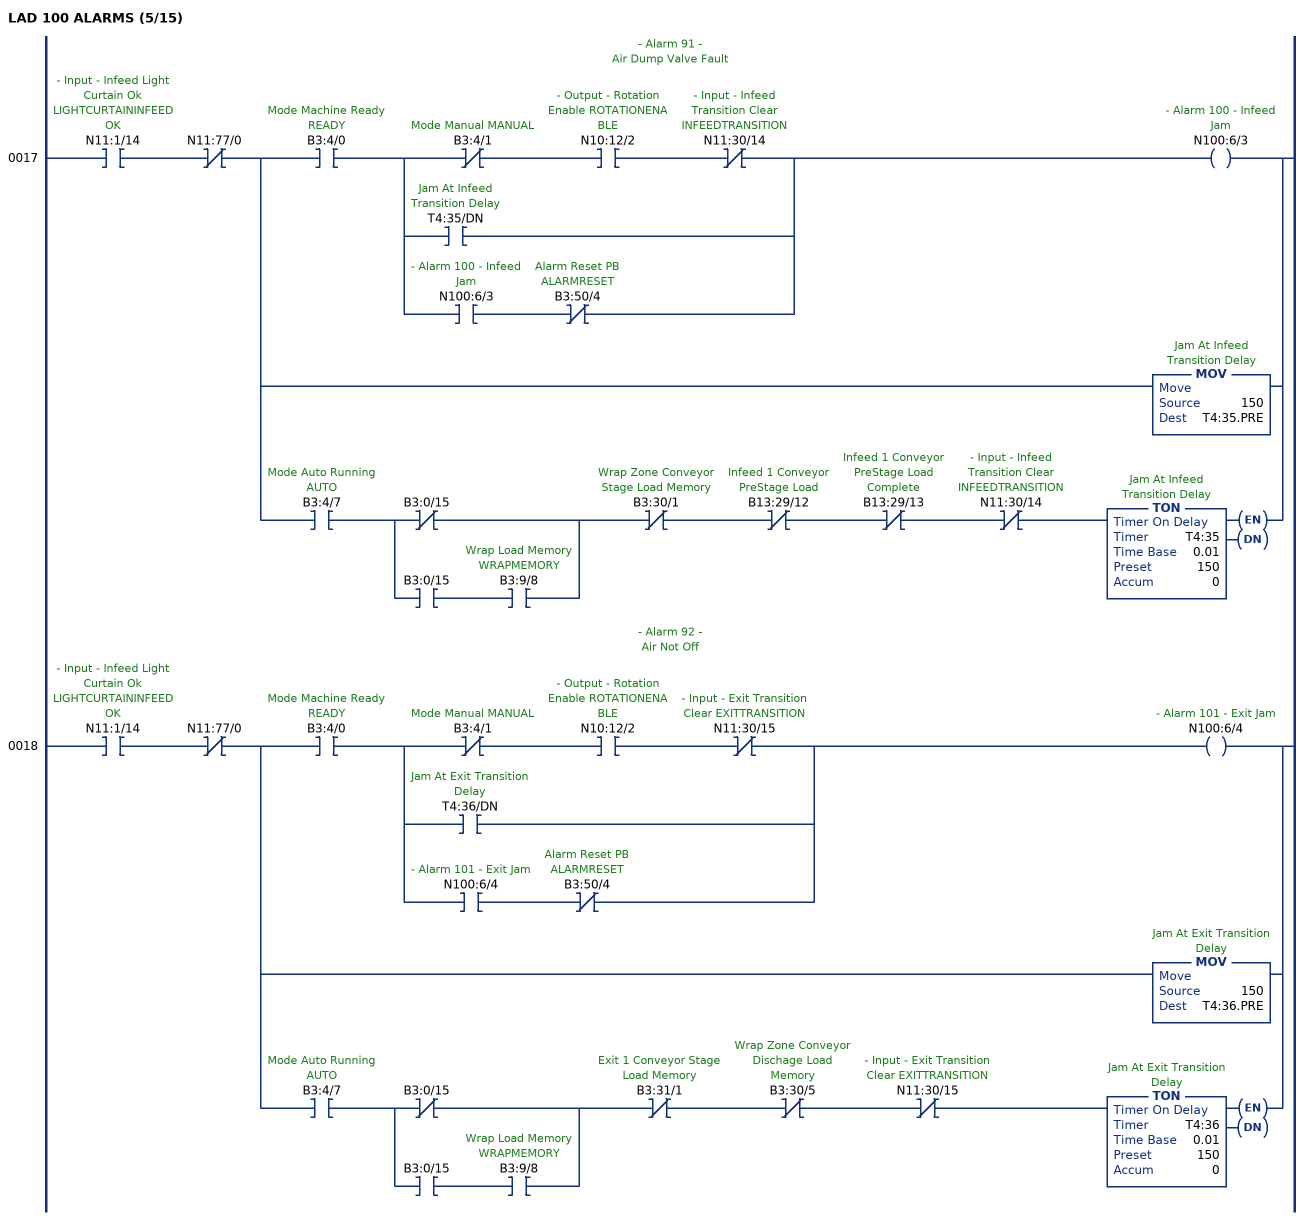
% Rung: 17 %
% - Alarm 91 -
% 
% Air Dump Valve Fault %
SOR XIC N11:1/14 XIO N11:77/0 BST XIC B3:4/0 BST XIO B3:4/1 XIC N10:12/2 XIO N11:30/14 NXB XIC T4:35/DN NXB XIC N100:6/3 XIO B3:50/4 BND OTE N100:6/3 NXB MOV 150 T4:35.PRE NXB XIC B3:4/7 BST XIO B3:0/15 NXB XIC B3:0/15 XIC B3:9/8 BND XIO B3:30/1 XIO B13:29/12 XIO B13:29/13 XIO N11:30/14 TON T4:35 0.01 150 0 BND EOR
%   N11:1/14  LIGHTCURTAININFEEDOK  "- Input - Infeed Light Curtain Ok" %
%   B3:4/0  READY  "Mode Machine Ready" %
%   B3:4/1  MANUAL  "Mode Manual" %
%   N10:12/2  ROTATIONENABLE  "- Output - Rotation Enable" %
%   N11:30/14  INFEEDTRANSITION  "- Input - Infeed Transition Clear" %
%   T4:35  "Jam At Infeed Transition Delay" %
%   N100:6/3  "- Alarm 100 - Infeed Jam" %
%   B3:50/4  ALARMRESET  "Alarm Reset PB" %
%   B3:4/7  AUTO  "Mode Auto Running" %
%   B3:9/8  WRAPMEMORY  "Wrap Load Memory" %
%   B3:30/1  "Wrap Zone Conveyor Stage Load Memory" %
%   B13:29/12  "Infeed 1 Conveyor PreStage Load" %
%   B13:29/13  "Infeed 1 Conveyor PreStage Load Complete" %
% Rung: 18 %
% - Alarm 92 -
% 
% Air Not Off %
SOR XIC N11:1/14 XIO N11:77/0 BST XIC B3:4/0 BST XIO B3:4/1 XIC N10:12/2 XIO N11:30/15 NXB XIC T4:36/DN NXB XIC N100:6/4 XIO B3:50/4 BND OTE N100:6/4 NXB MOV 150 T4:36.PRE NXB XIC B3:4/7 BST XIO B3:0/15 NXB XIC B3:0/15 XIC B3:9/8 BND XIO B3:31/1 XIO B3:30/5 XIO N11:30/15 TON T4:36 0.01 150 0 BND EOR
%   N11:1/14  LIGHTCURTAININFEEDOK  "- Input - Infeed Light Curtain Ok" %
%   B3:4/0  READY  "Mode Machine Ready" %
%   B3:4/1  MANUAL  "Mode Manual" %
%   N10:12/2  ROTATIONENABLE  "- Output - Rotation Enable" %
%   N11:30/15  EXITTRANSITION  "- Input - Exit Transition Clear" %
%   T4:36  "Jam At Exit Transition Delay" %
%   N100:6/4  "- Alarm 101 - Exit Jam" %
%   B3:50/4  ALARMRESET  "Alarm Reset PB" %
%   B3:4/7  AUTO  "Mode Auto Running" %
%   B3:9/8  WRAPMEMORY  "Wrap Load Memory" %
%   B3:31/1  "Exit 1 Conveyor Stage Load Memory" %
%   B3:30/5  "Wrap Zone Conveyor Dischage Load Memory" %

